LIN {X 0,Y 488.687,Z 319.919,A -85,B 0,C 180,E1 -6521.601,E2 -6521.601} C_VEL
LIN {X 0,Y 488.693,Z 319.925,A -85,B 0,C 180,E1 -6524.803,E2 -6524.803} C_VEL
LIN {X 0,Y 488.728,Z 319.952,A -85,B 0,C 180,E1 -6527.596,E2 -6527.596} C_VEL
LIN {X 0,Y 492.392,Z 332.248,A -85,B 0,C 180,E1 -6530.421,E2 -6530.421} C_VEL
LIN {X 0,Y 495.369,Z 342.536,A -85,B 0,C 180,E1 -6532.607,E2 -6532.607} C_VEL
LIN {X 0,Y 496.704,Z 348.362,A -85,B 0,C 180,E1 -6533.756,E2 -6533.756} C_VEL
LIN {X 0,Y 495.507,Z 364.581,A -85,B 0,C 180,E1 -6536.42,E2 -6536.42} C_VEL
LIN {X 0,Y 494.27,Z 383.903,A -85,B 0,C 180,E1 -6539.451,E2 -6539.451} C_VEL
LIN {X 0,Y 493.327,Z 401.965,A -85,B 0,C 180,E1 -6542.171,E2 -6542.171} C_VEL
LIN {X 0,Y 492.268,Z 420.732,A -85,B 0,C 180,E1 -6544.998,E2 -6544.998} C_VEL
LIN {X 0,Y 496.9,Z 441.839,A -85,B 0,C 180,E1 -6545.607,E2 -6545.607} C_VEL
LIN {X 0,Y 496.367,Z 458.327,A -85,B 0,C 180,E1 -6546.014,E2 -6546.014} C_VEL
LIN {X 0,Y 495.765,Z 473.338,A -85,B 0,C 180,E1 -6546.533,E2 -6546.533} C_VEL
LIN {X 0,Y 495.092,Z 488.171,A -85,B 0,C 180,E1 -6547.191,E2 -6547.191} C_VEL
LIN {X 0,Y 494.154,Z 504.481,A -85,B 0,C 180,E1 -6548.107,E2 -6548.107} C_VEL
LIN {X 0,Y 493.218,Z 519.301,A -85,B 0,C 180,E1 -6549.134,E2 -6549.134} C_VEL
LIN {X 0,Y 492.292,Z 533.052,A -85,B 0,C 180,E1 -6550.275,E2 -6550.275} C_VEL
LIN {X 0,Y 491.438,Z 545.141,A -85,B 0,C 180,E1 -6551.449,E2 -6551.449} C_VEL
LIN {X 0,Y 490.654,Z 556.299,A -85,B 0,C 180,E1 -6552.712,E2 -6552.712} C_VEL
LIN {X 0,Y 489.963,Z 567.437,A -85,B 0,C 180,E1 -6554.187,E2 -6554.187} C_VEL
LIN {X 0,Y 489.276,Z 578.223,A -85,B 0,C 180,E1 -6555.868,E2 -6555.868} C_VEL
LIN {X 0,Y 488.782,Z 587.283,A -85,B 0,C 180,E1 -6557.547,E2 -6557.547} C_VEL
LIN {X 0,Y 488.439,Z 594.861,A -85,B 0,C 180,E1 -6559.221,E2 -6559.221} C_VEL
LIN {X 0,Y 488.13,Z 602.47,A -85,B 0,C 180,E1 -6561.307,E2 -6561.307} C_VEL
LIN {X 0,Y 488.025,Z 608.25,A -85,B 0,C 180,E1 -6563.387,E2 -6563.387} C_VEL
LIN {X 0,Y 487.908,Z 611.638,A -85,B 0,C 180,E1 -6565.044,E2 -6565.044} C_VEL
LIN {X 0,Y 487.943,Z 614.092,A -85,B 0,C 180,E1 -6566.699,E2 -6566.699} C_VEL
LIN {X 0,Y 487.883,Z 615.48,A -85,B 0,C 180,E1 -6568.351,E2 -6568.351} C_VEL
LIN {X 0,Y 487.814,Z 616,A -85,B 0,C 180,E1 -6570.002,E2 -6570.002} C_VEL
LIN {X 0,Y 487.883,Z 615.477,A -85,B 0,C 180,E1 -6571.653,E2 -6571.653} C_VEL
LIN {X 0,Y 487.945,Z 614.087,A -85,B 0,C 180,E1 -6573.305,E2 -6573.305} C_VEL
LIN {X 0,Y 487.909,Z 611.631,A -85,B 0,C 180,E1 -6574.96,E2 -6574.96} C_VEL
LIN {X 0,Y 488.029,Z 608.246,A -85,B 0,C 180,E1 -6576.617,E2 -6576.617} C_VEL
LIN {X 0,Y 488.124,Z 602.462,A -85,B 0,C 180,E1 -6578.697,E2 -6578.697} C_VEL
LIN {X 0,Y 488.436,Z 594.848,A -85,B 0,C 180,E1 -6580.783,E2 -6580.783} C_VEL
LIN {X 0,Y 488.826,Z 586.246,A -85,B 0,C 180,E1 -6582.667,E2 -6582.667} C_VEL
LIN {X 0,Y 489.349,Z 576.967,A -85,B 0,C 180,E1 -6584.346,E2 -6584.346} C_VEL
LIN {X 0,Y 489.93,Z 567.409,A -85,B 0,C 180,E1 -6585.818,E2 -6585.818} C_VEL
LIN {X 0,Y 490.661,Z 556.269,A -85,B 0,C 180,E1 -6587.292,E2 -6587.292} C_VEL
LIN {X 0,Y 491.499,Z 544.123,A -85,B 0,C 180,E1 -6588.661,E2 -6588.661} C_VEL
LIN {X 0,Y 492.423,Z 530.761,A -85,B 0,C 180,E1 -6589.932,E2 -6589.932} C_VEL
LIN {X 0,Y 493.327,Z 517.822,A -85,B 0,C 180,E1 -6590.975,E2 -6590.975} C_VEL
LIN {X 0,Y 494.159,Z 504.385,A -85,B 0,C 180,E1 -6591.899,E2 -6591.899} C_VEL
LIN {X 0,Y 495.108,Z 488.383,A -85,B 0,C 180,E1 -6592.796,E2 -6592.796} C_VEL
LIN {X 0,Y 495.69,Z 475.201,A -85,B 0,C 180,E1 -6593.392,E2 -6593.392} C_VEL
LIN {X 0,Y 496.355,Z 458.459,A -85,B 0,C 180,E1 -6593.983,E2 -6593.983} C_VEL
LIN {X 0,Y 496.893,Z 442.168,A -85,B 0,C 180,E1 -6594.387,E2 -6594.387} C_VEL
LIN {X 0,Y 493.328,Z 425.29,A -85,B 0,C 180,E1 -6594.865,E2 -6594.865} C_VEL
LIN {X 0,Y 492.313,Z 420.685,A -85,B 0,C 180,E1 -6595.006,E2 -6595.006} C_VEL
LIN {X 0,Y 493.312,Z 402.026,A -85,B 0,C 180,E1 -6597.821,E2 -6597.821} C_VEL
LIN {X 0,Y 494.313,Z 382.243,A -85,B 0,C 180,E1 -6600.788,E2 -6600.788} C_VEL
LIN {X 0,Y 495.292,Z 365.983,A -85,B 0,C 180,E1 -6603.29,E2 -6603.29} C_VEL
LIN {X 0,Y 496.841,Z 349.707,A -85,B 0,C 180,E1 -6606.095,E2 -6606.095} C_VEL
LIN {X 0,Y 496.561,Z 346.659,A -85,B 0,C 180,E1 -6606.719,E2 -6606.719} C_VEL
LIN {X 0,Y 494.656,Z 338.928,A -85,B 0,C 180,E1 -6608.609,E2 -6608.609} C_VEL
LIN {X 0,Y 492.734,Z 332.835,A -85,B 0,C 180,E1 -6610.481,E2 -6610.481} C_VEL
LIN {X 0,Y 491.301,Z 328.379,A -85,B 0,C 180,E1 -6612.249,E2 -6612.249} C_VEL
LIN {X 0,Y 490.173,Z 324.874,A -85,B 0,C 180,E1 -6614.202,E2 -6614.202} C_VEL
LIN {X 0,Y 489.577,Z 323.156,A -85,B 0,C 180,E1 -6615.872,E2 -6615.872} C_VEL
LIN {X 0,Y 489.411,Z 322.532,A -85,B 0,C 180,E1 -6617.552,E2 -6617.552} C_VEL
LIN {X 0,Y 489.532,Z 323.246,A -85,B 0,C 180,E1 -6619.545,E2 -6619.545} C_VEL
LIN {X 0,Y 489.855,Z 324.388,A -85,B 0,C 180,E1 -6620.856,E2 -6620.856} C_VEL
LIN {X 0,Y 490.458,Z 327.705,A -85,B 0,C 180,E1 -6623.366,E2 -6623.366} C_VEL
LIN {X 0,Y 490.697,Z 330.547,A -85,B 0,C 180,E1 -6625.048,E2 -6625.048} C_VEL
LIN {X 0,Y 490.306,Z 335.636,A -85,B 0,C 180,E1 -6627.749,E2 -6627.749} C_VEL
LIN {X 0,Y 489.938,Z 341.889,A -85,B 0,C 180,E1 -6631.05,E2 -6631.05} C_VEL
LIN {X 0,Y 489.753,Z 346.67,A -85,B 0,C 180,E1 -6633.586,E2 -6633.586} C_VEL
LIN {X 0,Y 489.517,Z 352.555,A -85,B 0,C 180,E1 -6636.76,E2 -6636.76} C_VEL
LIN {X 0,Y 489.316,Z 358.293,A -85,B 0,C 180,E1 -6639.836,E2 -6639.836} C_VEL
LIN {X 0,Y 489.109,Z 363.152,A -85,B 0,C 180,E1 -6642.438,E2 -6642.438} C_VEL
LIN {X 0,Y 489.022,Z 367.71,A -85,B 0,C 180,E1 -6644.846,E2 -6644.846} C_VEL
LIN {X 0,Y 492.349,Z 378.298,A -85,B 0,C 180,E1 -6645.323,E2 -6645.323} C_VEL
LIN {X 0,Y 491.939,Z 392.152,A -85,B 0,C 180,E1 -6645.892,E2 -6645.892} C_VEL
LIN {X 0,Y 491.362,Z 405.497,A -85,B 0,C 180,E1 -6646.634,E2 -6646.634} C_VEL
LIN {X 0,Y 490.964,Z 417.712,A -85,B 0,C 180,E1 -6647.515,E2 -6647.515} C_VEL
LIN {X 0,Y 490.431,Z 428.93,A -85,B 0,C 180,E1 -6648.532,E2 -6648.532} C_VEL
LIN {X 0,Y 490.077,Z 439.066,A -85,B 0,C 180,E1 -6649.674,E2 -6649.674} C_VEL
LIN {X 0,Y 489.619,Z 447.947,A -85,B 0,C 180,E1 -6650.916,E2 -6650.916} C_VEL
LIN {X 0,Y 489.345,Z 454.492,A -85,B 0,C 180,E1 -6652.044,E2 -6652.044} C_VEL
LIN {X 0,Y 489.014,Z 460.816,A -85,B 0,C 180,E1 -6653.398,E2 -6653.398} C_VEL
LIN {X 0,Y 488.814,Z 465.319,A -85,B 0,C 180,E1 -6654.638,E2 -6654.638} C_VEL
LIN {X 0,Y 488.754,Z 468.722,A -85,B 0,C 180,E1 -6655.877,E2 -6655.877} C_VEL
LIN {X 0,Y 488.686,Z 470.465,A -85,B 0,C 180,E1 -6656.703,E2 -6656.703} C_VEL
LIN {X 0,Y 488.565,Z 471.782,A -85,B 0,C 180,E1 -6657.527,E2 -6657.527} C_VEL
LIN {X 0,Y 488.377,Z 473.181,A -85,B 0,C 180,E1 -6659.176,E2 -6659.176} C_VEL
LIN {X 0,Y 488.357,Z 473.297,A -85,B 0,C 180,E1 -6660,E2 -6660} C_VEL
LIN {X 0,Y 488.366,Z 473.016,A -85,B 0,C 180,E1 -6660.825,E2 -6660.825} C_VEL
LIN {X 0,Y 488.43,Z 472.307,A -85,B 0,C 180,E1 -6661.649,E2 -6661.649} C_VEL
LIN {X 0,Y 488.431,Z 471.22,A -85,B 0,C 180,E1 -6662.474,E2 -6662.474} C_VEL
LIN {X 0,Y 488.547,Z 469.723,A -85,B 0,C 180,E1 -6663.299,E2 -6663.299} C_VEL
LIN {X 0,Y 488.513,Z 466.692,A -85,B 0,C 180,E1 -6664.539,E2 -6664.539} C_VEL
LIN {X 0,Y 488.635,Z 462.622,A -85,B 0,C 180,E1 -6665.779,E2 -6665.779} C_VEL
LIN {X 0,Y 488.827,Z 456.426,A -85,B 0,C 180,E1 -6667.232,E2 -6667.232} C_VEL
LIN {X 0,Y 489.088,Z 449.68,A -85,B 0,C 180,E1 -6668.47,E2 -6668.47} C_VEL
LIN {X 0,Y 489.342,Z 441.317,A -85,B 0,C 180,E1 -6669.716,E2 -6669.716} C_VEL
LIN {X 0,Y 489.638,Z 432.812,A -85,B 0,C 180,E1 -6670.754,E2 -6670.754} C_VEL
LIN {X 0,Y 490.038,Z 422.438,A -85,B 0,C 180,E1 -6671.793,E2 -6671.793} C_VEL
LIN {X 0,Y 490.401,Z 411.409,A -85,B 0,C 180,E1 -6672.684,E2 -6672.684} C_VEL
LIN {X 0,Y 490.868,Z 399.455,A -85,B 0,C 180,E1 -6673.454,E2 -6673.454} C_VEL
LIN {X 0,Y 491.139,Z 386.946,A -85,B 0,C 180,E1 -6674.08,E2 -6674.08} C_VEL
LIN {X 0,Y 491.244,Z 376.285,A -85,B 0,C 180,E1 -6674.486,E2 -6674.486} C_VEL
LIN {X 0,Y 488.33,Z 363.648,A -85,B 0,C 180,E1 -6674.934,E2 -6674.934} C_VEL
LIN {X 0,Y 488.388,Z 356.44,A -85,B 0,C 180,E1 -6678.457,E2 -6678.457} C_VEL
LIN {X 0,Y 488.55,Z 349.357,A -85,B 0,C 180,E1 -6681.964,E2 -6681.964} C_VEL
LIN {X 0,Y 488.661,Z 343.202,A -85,B 0,C 180,E1 -6685.029,E2 -6685.029} C_VEL
LIN {X 0,Y 488.725,Z 338.504,A -85,B 0,C 180,E1 -6687.398,E2 -6687.398} C_VEL
LIN {X 0,Y 488.885,Z 332.597,A -85,B 0,C 180,E1 -6690.396,E2 -6690.396} C_VEL
LIN {X 0,Y 489.043,Z 326.458,A -85,B 0,C 180,E1 -6693.537,E2 -6693.537} C_VEL
LIN {X 0,Y 488.964,Z 321.505,A -85,B 0,C 180,E1 -6696.108,E2 -6696.108} C_VEL
LIN {X 0,Y 488.712,Z 319.925,A -85,B 0,C 180,E1 -6697.052,E2 -6697.052} C_VEL
LIN {X 0,Y 488.727,Z 319.923,A -85,B 0,C 180,E1 -6700.344,E2 -6700.344} C_VEL
LIN {X 0,Y 488.686,Z 319.926,A -85,B 0,C 180,E1 -6703.655,E2 -6703.655} C_VEL
LIN {X 0,Y 488.685,Z 319.927,A -85,B 0,C 180,E1 -6706.344,E2 -6706.344} C_VEL
LIN {X 0,Y 488.712,Z 319.922,A -85,B 0,C 180,E1 -6709.673,E2 -6709.673} C_VEL
LIN {X 0,Y 488.696,Z 319.928,A -85,B 0,C 180,E1 -6712.841,E2 -6712.841} C_VEL
LIN {X 0,Y 488.785,Z 320.145,A -85,B 0,C 180,E1 -6713.49,E2 -6713.49} C_VEL
LIN {X 0,Y 489.294,Z 324.961,A -85,B 0,C 180,E1 -6715.451,E2 -6715.451} C_VEL
LIN {X 0,Y 489.247,Z 329.472,A -85,B 0,C 180,E1 -6717.377,E2 -6717.377} C_VEL
LIN {X 0,Y 488.584,Z 331.063,A -85,B 0,C 180,E1 -6718.038,E2 -6718.038} C_VEL
LIN {X 0,Y 485.698,Z 333.904,A -85,B 0,C 180,E1 -6719.103,E2 -6719.103} C_VEL
LIN {X 0,Y 483.247,Z 336.161,A -85,B 0,C 180,E1 -6719.961,E2 -6719.961} C_VEL
LIN {X 0,Y 482.19,Z 337.745,A -85,B 0,C 180,E1 -6720.63,E2 -6720.63} C_VEL
LIN {X 0,Y 482.103,Z 338.23,A -85,B 0,C 180,E1 -6720.858,E2 -6720.858} C_VEL
LIN {X 0,Y 481.968,Z 344.726,A -85,B 0,C 180,E1 -6724.057,E2 -6724.057} C_VEL
LIN {X 0,Y 481.938,Z 350.288,A -85,B 0,C 180,E1 -6726.811,E2 -6726.811} C_VEL
LIN {X 0,Y 481.835,Z 355.858,A -85,B 0,C 180,E1 -6729.507,E2 -6729.507} C_VEL
LIN {X 0,Y 481.786,Z 362.714,A -85,B 0,C 180,E1 -6732.598,E2 -6732.598} C_VEL
LIN {X 0,Y 481.935,Z 369.073,A -85,B 0,C 180,E1 -6735.145,E2 -6735.145} C_VEL
LIN {X 0,Y 484.514,Z 378.706,A -85,B 0,C 180,E1 -6735.462,E2 -6735.462} C_VEL
LIN {X 0,Y 484.31,Z 391.761,A -85,B 0,C 180,E1 -6735.931,E2 -6735.931} C_VEL
LIN {X 0,Y 483.99,Z 404.316,A -85,B 0,C 180,E1 -6736.564,E2 -6736.564} C_VEL
LIN {X 0,Y 483.777,Z 415.235,A -85,B 0,C 180,E1 -6737.293,E2 -6737.293} C_VEL
LIN {X 0,Y 483.401,Z 425.434,A -85,B 0,C 180,E1 -6738.148,E2 -6738.148} C_VEL
LIN {X 0,Y 482.991,Z 434.651,A -85,B 0,C 180,E1 -6739.094,E2 -6739.094} C_VEL
LIN {X 0,Y 482.672,Z 443.053,A -85,B 0,C 180,E1 -6740.147,E2 -6740.147} C_VEL
LIN {X 0,Y 482.284,Z 451.234,A -85,B 0,C 180,E1 -6741.408,E2 -6741.408} C_VEL
LIN {X 0,Y 481.965,Z 457.873,A -85,B 0,C 180,E1 -6742.692,E2 -6742.692} C_VEL
LIN {X 0,Y 481.743,Z 463.73,A -85,B 0,C 180,E1 -6744.137,E2 -6744.137} C_VEL
LIN {X 0,Y 481.532,Z 467.616,A -85,B 0,C 180,E1 -6745.394,E2 -6745.394} C_VEL
LIN {X 0,Y 481.453,Z 470.471,A -85,B 0,C 180,E1 -6746.651,E2 -6746.651} C_VEL
LIN {X 0,Y 481.419,Z 471.858,A -85,B 0,C 180,E1 -6747.488,E2 -6747.488} C_VEL
LIN {X 0,Y 481.352,Z 473.433,A -85,B 0,C 180,E1 -6749.161,E2 -6749.161} C_VEL
LIN {X 0,Y 481.337,Z 473.667,A -85,B 0,C 180,E1 -6749.998,E2 -6749.998} C_VEL
LIN {X 0,Y 481.351,Z 473.484,A -85,B 0,C 180,E1 -6750.835,E2 -6750.835} C_VEL
LIN {X 0,Y 481.294,Z 472.929,A -85,B 0,C 180,E1 -6751.671,E2 -6751.671} C_VEL
LIN {X 0,Y 481.558,Z 470.64,A -85,B 0,C 180,E1 -6753.345,E2 -6753.345} C_VEL
LIN {X 0,Y 481.622,Z 467.856,A -85,B 0,C 180,E1 -6754.601,E2 -6754.601} C_VEL
LIN {X 0,Y 481.733,Z 464.067,A -85,B 0,C 180,E1 -6755.859,E2 -6755.859} C_VEL
LIN {X 0,Y 481.879,Z 459.586,A -85,B 0,C 180,E1 -6757.019,E2 -6757.019} C_VEL
LIN {X 0,Y 482.197,Z 452.93,A -85,B 0,C 180,E1 -6758.378,E2 -6758.378} C_VEL
LIN {X 0,Y 482.586,Z 445.185,A -85,B 0,C 180,E1 -6759.639,E2 -6759.639} C_VEL
LIN {X 0,Y 482.9,Z 437.274,A -85,B 0,C 180,E1 -6760.691,E2 -6760.691} C_VEL
LIN {X 0,Y 483.287,Z 427.556,A -85,B 0,C 180,E1 -6761.745,E2 -6761.745} C_VEL
LIN {X 0,Y 483.605,Z 417.954,A -85,B 0,C 180,E1 -6762.589,E2 -6762.589} C_VEL
LIN {X 0,Y 483.943,Z 405.879,A -85,B 0,C 180,E1 -6763.434,E2 -6763.434} C_VEL
LIN {X 0,Y 484.272,Z 393.904,A -85,B 0,C 180,E1 -6764.066,E2 -6764.066} C_VEL
LIN {X 0,Y 484.476,Z 380.633,A -85,B 0,C 180,E1 -6764.57,E2 -6764.57} C_VEL
LIN {X 0,Y 484.196,Z 377.035,A -85,B 0,C 180,E1 -6764.684,E2 -6764.684} C_VEL
LIN {X 0,Y 481.89,Z 368.836,A -85,B 0,C 180,E1 -6764.974,E2 -6764.974} C_VEL
LIN {X 0,Y 481.776,Z 361.933,A -85,B 0,C 180,E1 -6767.836,E2 -6767.836} C_VEL
LIN {X 0,Y 481.85,Z 354.941,A -85,B 0,C 180,E1 -6771.017,E2 -6771.017} C_VEL
LIN {X 0,Y 481.946,Z 348.668,A -85,B 0,C 180,E1 -6774.096,E2 -6774.096} C_VEL
LIN {X 0,Y 482.04,Z 342.372,A -85,B 0,C 180,E1 -6777.206,E2 -6777.206} C_VEL
LIN {X 0,Y 482.189,Z 336.25,A -85,B 0,C 180,E1 -6780.185,E2 -6780.185} C_VEL
LIN {X 0,Y 482.285,Z 329.836,A -85,B 0,C 180,E1 -6783.121,E2 -6783.121} C_VEL
LIN {X 0,Y 482.199,Z 323.807,A -85,B 0,C 180,E1 -6785.658,E2 -6785.658} C_VEL
LIN {X 0,Y 481.7,Z 320.8,A -85,B 0,C 180,E1 -6786.867,E2 -6786.867} C_VEL
LIN {X 0,Y 481.646,Z 320.805,A -85,B 0,C 180,E1 -6789.94,E2 -6789.94} C_VEL
LIN {X 0,Y 481.613,Z 320.808,A -85,B 0,C 180,E1 -6793.144,E2 -6793.144} C_VEL
LIN {X 0,Y 481.644,Z 320.801,A -85,B 0,C 180,E1 -6795.638,E2 -6795.638} C_VEL
LIN {X 0,Y 481.66,Z 320.798,A -85,B 0,C 180,E1 -6798.082,E2 -6798.082} C_VEL
LIN {X 0,Y 481.689,Z 320.794,A -85,B 0,C 180,E1 -6801.142,E2 -6801.142} C_VEL
LIN {X 0,Y 481.648,Z 320.799,A -85,B 0,C 180,E1 -6804.793,E2 -6804.793} C_VEL
LIN {X 0,Y 481.652,Z 320.802,A -85,B 0,C 180,E1 -6807.324,E2 -6807.324} C_VEL
LIN {X 0,Y 481.658,Z 320.796,A -85,B 0,C 180,E1 -6810.257,E2 -6810.257} C_VEL
LIN {X 0,Y 481.731,Z 320.786,A -85,B 0,C 180,E1 -6813.111,E2 -6813.111} C_VEL
LIN {X 0,Y 481.672,Z 320.8,A -85,B 0,C 180,E1 -6815.886,E2 -6815.886} C_VEL
LIN {X 0,Y 481.688,Z 320.795,A -85,B 0,C 180,E1 -6819.023,E2 -6819.023} C_VEL
LIN {X 0,Y 481.682,Z 320.793,A -85,B 0,C 180,E1 -6822.157,E2 -6822.157} C_VEL
LIN {X 0,Y 481.718,Z 320.793,A -85,B 0,C 180,E1 -6824.775,E2 -6824.775} C_VEL
LIN {X 0,Y 481.777,Z 320.787,A -85,B 0,C 180,E1 -6828.215,E2 -6828.215} C_VEL
LIN {X 0,Y 481.747,Z 320.786,A -85,B 0,C 180,E1 -6831.611,E2 -6831.611} C_VEL
LIN {X 0,Y 481.797,Z 320.779,A -85,B 0,C 180,E1 -6834.139,E2 -6834.139} C_VEL
LIN {X 0,Y 481.898,Z 320.77,A -85,B 0,C 180,E1 -6837.492,E2 -6837.492} C_VEL
LIN {X 0,Y 481.902,Z 320.766,A -85,B 0,C 180,E1 -6840.835,E2 -6840.835} C_VEL
LIN {X 0,Y 481.912,Z 320.771,A -85,B 0,C 180,E1 -6842.507,E2 -6842.507} C_VEL
LIN {X 0,Y 481.809,Z 320.785,A -85,B 0,C 180,E1 -6845.86,E2 -6845.86} C_VEL
LIN {X 0,Y 481.739,Z 320.788,A -85,B 0,C 180,E1 -6848.388,E2 -6848.388} C_VEL
LIN {X 0,Y 481.772,Z 320.785,A -85,B 0,C 180,E1 -6851.784,E2 -6851.784} C_VEL
LIN {X 0,Y 481.718,Z 320.791,A -85,B 0,C 180,E1 -6855.225,E2 -6855.225} C_VEL
LIN {X 0,Y 481.693,Z 320.794,A -85,B 0,C 180,E1 -6858.722,E2 -6858.722} C_VEL
LIN {X 0,Y 481.654,Z 320.803,A -85,B 0,C 180,E1 -6861.394,E2 -6861.394} C_VEL
LIN {X 0,Y 481.665,Z 320.797,A -85,B 0,C 180,E1 -6864.113,E2 -6864.113} C_VEL
LIN {X 0,Y 481.722,Z 320.792,A -85,B 0,C 180,E1 -6867.14,E2 -6867.14} C_VEL
LIN {X 0,Y 481.655,Z 320.799,A -85,B 0,C 180,E1 -6869.742,E2 -6869.742} C_VEL
LIN {X 0,Y 481.651,Z 320.8,A -85,B 0,C 180,E1 -6872.675,E2 -6872.675} C_VEL
LIN {X 0,Y 481.623,Z 320.807,A -85,B 0,C 180,E1 -6875.71,E2 -6875.71} C_VEL
LIN {X 0,Y 481.651,Z 320.802,A -85,B 0,C 180,E1 -6878.861,E2 -6878.861} C_VEL
LIN {X 0,Y 481.632,Z 320.799,A -85,B 0,C 180,E1 -6881.915,E2 -6881.915} C_VEL
LIN {X 0,Y 481.641,Z 320.805,A -85,B 0,C 180,E1 -6884.459,E2 -6884.459} C_VEL
LIN {X 0,Y 481.701,Z 320.949,A -85,B 0,C 180,E1 -6886.997,E2 -6886.997} C_VEL
LIN {X 0,Y 484.936,Z 331.574,A -85,B 0,C 180,E1 -6889.539,E2 -6889.539} C_VEL
LIN {X 0,Y 488.601,Z 344.148,A -85,B 0,C 180,E1 -6892.289,E2 -6892.289} C_VEL
LIN {X 0,Y 490.108,Z 350.895,A -85,B 0,C 180,E1 -6893.648,E2 -6893.648} C_VEL
LIN {X 0,Y 488.612,Z 369.086,A -85,B 0,C 180,E1 -6896.672,E2 -6896.672} C_VEL
LIN {X 0,Y 487.34,Z 388.12,A -85,B 0,C 180,E1 -6899.689,E2 -6899.689} C_VEL
LIN {X 0,Y 486.277,Z 407.911,A -85,B 0,C 180,E1 -6902.689,E2 -6902.689} C_VEL
LIN {X 0,Y 485.554,Z 420.739,A -85,B 0,C 180,E1 -6904.629,E2 -6904.629} C_VEL
LIN {X 0,Y 490.394,Z 442.388,A -85,B 0,C 180,E1 -6905.272,E2 -6905.272} C_VEL
LIN {X 0,Y 489.844,Z 459.443,A -85,B 0,C 180,E1 -6905.709,E2 -6905.709} C_VEL
LIN {X 0,Y 489.146,Z 475.3,A -85,B 0,C 180,E1 -6906.281,E2 -6906.281} C_VEL
LIN {X 0,Y 488.382,Z 489.912,A -85,B 0,C 180,E1 -6906.958,E2 -6906.958} C_VEL
LIN {X 0,Y 487.538,Z 504.667,A -85,B 0,C 180,E1 -6907.806,E2 -6907.806} C_VEL
LIN {X 0,Y 486.544,Z 519.299,A -85,B 0,C 180,E1 -6908.834,E2 -6908.834} C_VEL
LIN {X 0,Y 485.608,Z 532.128,A -85,B 0,C 180,E1 -6909.905,E2 -6909.905} C_VEL
LIN {X 0,Y 484.731,Z 544.166,A -85,B 0,C 180,E1 -6911.073,E2 -6911.073} C_VEL
LIN {X 0,Y 483.78,Z 556.299,A -85,B 0,C 180,E1 -6912.458,E2 -6912.458} C_VEL
LIN {X 0,Y 483.031,Z 567.437,A -85,B 0,C 180,E1 -6913.954,E2 -6913.954} C_VEL
LIN {X 0,Y 482.3,Z 578.222,A -85,B 0,C 180,E1 -6915.66,E2 -6915.66} C_VEL
LIN {X 0,Y 481.741,Z 587.284,A -85,B 0,C 180,E1 -6917.362,E2 -6917.362} C_VEL
LIN {X 0,Y 481.413,Z 594.86,A -85,B 0,C 180,E1 -6919.062,E2 -6919.062} C_VEL
LIN {X 0,Y 481.063,Z 602.47,A -85,B 0,C 180,E1 -6921.178,E2 -6921.178} C_VEL
LIN {X 0,Y 480.948,Z 608.25,A -85,B 0,C 180,E1 -6923.289,E2 -6923.289} C_VEL
LIN {X 0,Y 480.834,Z 611.638,A -85,B 0,C 180,E1 -6924.971,E2 -6924.971} C_VEL
LIN {X 0,Y 480.849,Z 614.092,A -85,B 0,C 180,E1 -6926.651,E2 -6926.651} C_VEL
LIN {X 0,Y 480.784,Z 615.48,A -85,B 0,C 180,E1 -6928.327,E2 -6928.327} C_VEL
LIN {X 0,Y 480.738,Z 616,A -85,B 0,C 180,E1 -6930.002,E2 -6930.002} C_VEL
LIN {X 0,Y 480.784,Z 615.477,A -85,B 0,C 180,E1 -6931.677,E2 -6931.677} C_VEL
LIN {X 0,Y 480.85,Z 614.087,A -85,B 0,C 180,E1 -6933.354,E2 -6933.354} C_VEL
LIN {X 0,Y 480.836,Z 611.631,A -85,B 0,C 180,E1 -6935.033,E2 -6935.033} C_VEL
LIN {X 0,Y 480.952,Z 608.247,A -85,B 0,C 180,E1 -6936.715,E2 -6936.715} C_VEL
LIN {X 0,Y 481.058,Z 602.462,A -85,B 0,C 180,E1 -6938.826,E2 -6938.826} C_VEL
LIN {X 0,Y 481.402,Z 594.848,A -85,B 0,C 180,E1 -6940.942,E2 -6940.942} C_VEL
LIN {X 0,Y 481.824,Z 586.247,A -85,B 0,C 180,E1 -6942.854,E2 -6942.854} C_VEL
LIN {X 0,Y 482.368,Z 576.967,A -85,B 0,C 180,E1 -6944.558,E2 -6944.558} C_VEL
LIN {X 0,Y 483,Z 567.409,A -85,B 0,C 180,E1 -6946.051,E2 -6946.051} C_VEL
LIN {X 0,Y 483.786,Z 556.269,A -85,B 0,C 180,E1 -6947.546,E2 -6947.546} C_VEL
LIN {X 0,Y 484.705,Z 544.122,A -85,B 0,C 180,E1 -6948.933,E2 -6948.933} C_VEL
LIN {X 0,Y 485.671,Z 530.857,A -85,B 0,C 180,E1 -6950.212,E2 -6950.212} C_VEL
LIN {X 0,Y 486.729,Z 516.394,A -85,B 0,C 180,E1 -6951.384,E2 -6951.384} C_VEL
LIN {X 0,Y 487.643,Z 503.092,A -85,B 0,C 180,E1 -6952.289,E2 -6952.289} C_VEL
LIN {X 0,Y 488.535,Z 488.381,A -85,B 0,C 180,E1 -6953.12,E2 -6953.12} C_VEL
LIN {X 0,Y 489.187,Z 475.201,A -85,B 0,C 180,E1 -6953.722,E2 -6953.722} C_VEL
LIN {X 0,Y 489.855,Z 459.341,A -85,B 0,C 180,E1 -6954.294,E2 -6954.294} C_VEL
LIN {X 0,Y 490.371,Z 443.722,A -85,B 0,C 180,E1 -6954.698,E2 -6954.698} C_VEL
LIN {X 0,Y 489.839,Z 439.91,A -85,B 0,C 180,E1 -6954.805,E2 -6954.805} C_VEL
LIN {X 0,Y 485.581,Z 420.702,A -85,B 0,C 180,E1 -6955.375,E2 -6955.375} C_VEL
LIN {X 0,Y 486.361,Z 404.997,A -85,B 0,C 180,E1 -6957.721,E2 -6957.721} C_VEL
LIN {X 0,Y 487.052,Z 391.301,A -85,B 0,C 180,E1 -6959.748,E2 -6959.748} C_VEL
LIN {X 0,Y 488.439,Z 369.736,A -85,B 0,C 180,E1 -6963.147,E2 -6963.147} C_VEL
LIN {X 0,Y 489.905,Z 354.515,A -85,B 0,C 180,E1 -6965.775,E2 -6965.775} C_VEL
LIN {X 0,Y 490.21,Z 350.269,A -85,B 0,C 180,E1 -6966.597,E2 -6966.597} C_VEL
LIN {X 0,Y 488.486,Z 342.788,A -85,B 0,C 180,E1 -6968.431,E2 -6968.431} C_VEL
LIN {X 0,Y 486.344,Z 335.866,A -85,B 0,C 180,E1 -6970.564,E2 -6970.564} C_VEL
LIN {X 0,Y 484.928,Z 331.462,A -85,B 0,C 180,E1 -6972.343,E2 -6972.343} C_VEL
LIN {X 0,Y 483.912,Z 328.176,A -85,B 0,C 180,E1 -6974.198,E2 -6974.198} C_VEL
LIN {X 0,Y 483.298,Z 326.493,A -85,B 0,C 180,E1 -6975.733,E2 -6975.733} C_VEL
LIN {X 0,Y 483.114,Z 325.812,A -85,B 0,C 180,E1 -6976.865,E2 -6976.865} C_VEL
LIN {X 0,Y 483.014,Z 325.651,A -85,B 0,C 180,E1 -6977.986,E2 -6977.986} C_VEL
LIN {X 0,Y 483.172,Z 326.576,A -85,B 0,C 180,E1 -6980.208,E2 -6980.208} C_VEL
LIN {X 0,Y 483.566,Z 328.817,A -85,B 0,C 180,E1 -6982.381,E2 -6982.381} C_VEL
LIN {X 0,Y 483.943,Z 331.868,A -85,B 0,C 180,E1 -6984.487,E2 -6984.487} C_VEL
LIN {X 0,Y 483.737,Z 335.341,A -85,B 0,C 180,E1 -6986.49,E2 -6986.49} C_VEL
LIN {X 0,Y 483.147,Z 342.416,A -85,B 0,C 180,E1 -6990.359,E2 -6990.359} C_VEL
LIN {X 0,Y 482.872,Z 347.642,A -85,B 0,C 180,E1 -6993.18,E2 -6993.18} C_VEL
LIN {X 0,Y 482.651,Z 352.751,A -85,B 0,C 180,E1 -6995.939,E2 -6995.939} C_VEL
LIN {X 0,Y 482.478,Z 357.918,A -85,B 0,C 180,E1 -6998.791,E2 -6998.791} C_VEL
LIN {X 0,Y 482.256,Z 362.567,A -85,B 0,C 180,E1 -7001.311,E2 -7001.311} C_VEL
LIN {X 0,Y 482.107,Z 368.73,A -85,B 0,C 180,E1 -7004.538,E2 -7004.538} C_VEL
LIN {X 0,Y 485.615,Z 379.619,A -85,B 0,C 180,E1 -7005.061,E2 -7005.061} C_VEL
LIN {X 0,Y 485.266,Z 393.198,A -85,B 0,C 180,E1 -7005.64,E2 -7005.64} C_VEL
LIN {X 0,Y 484.691,Z 405.834,A -85,B 0,C 180,E1 -7006.351,E2 -7006.351} C_VEL
LIN {X 0,Y 484.232,Z 418.091,A -85,B 0,C 180,E1 -7007.239,E2 -7007.239} C_VEL
LIN {X 0,Y 483.759,Z 428.36,A -85,B 0,C 180,E1 -7008.159,E2 -7008.159} C_VEL
LIN {X 0,Y 483.314,Z 438.752,A -85,B 0,C 180,E1 -7009.316,E2 -7009.316} C_VEL
LIN {X 0,Y 482.831,Z 447.947,A -85,B 0,C 180,E1 -7010.576,E2 -7010.576} C_VEL
LIN {X 0,Y 482.466,Z 455.669,A -85,B 0,C 180,E1 -7011.905,E2 -7011.905} C_VEL
LIN {X 0,Y 482.081,Z 462.108,A -85,B 0,C 180,E1 -7013.303,E2 -7013.303} C_VEL
LIN {X 0,Y 481.874,Z 466.596,A -85,B 0,C 180,E1 -7014.56,E2 -7014.56} C_VEL
LIN {X 0,Y 481.796,Z 469.986,A -85,B 0,C 180,E1 -7015.818,E2 -7015.818} C_VEL
LIN {X 0,Y 481.718,Z 471.714,A -85,B 0,C 180,E1 -7016.655,E2 -7016.655} C_VEL
LIN {X 0,Y 481.581,Z 473.018,A -85,B 0,C 180,E1 -7017.491,E2 -7017.491} C_VEL
LIN {X 0,Y 481.382,Z 474.388,A -85,B 0,C 180,E1 -7019.164,E2 -7019.164} C_VEL
LIN {X 0,Y 481.358,Z 474.487,A -85,B 0,C 180,E1 -7020,E2 -7020} C_VEL
LIN {X 0,Y 481.364,Z 474.18,A -85,B 0,C 180,E1 -7020.837,E2 -7020.837} C_VEL
LIN {X 0,Y 481.431,Z 473.445,A -85,B 0,C 180,E1 -7021.673,E2 -7021.673} C_VEL
LIN {X 0,Y 481.429,Z 472.338,A -85,B 0,C 180,E1 -7022.51,E2 -7022.51} C_VEL
LIN {X 0,Y 481.555,Z 470.819,A -85,B 0,C 180,E1 -7023.347,E2 -7023.347} C_VEL
LIN {X 0,Y 481.512,Z 467.75,A -85,B 0,C 180,E1 -7024.605,E2 -7024.605} C_VEL
LIN {X 0,Y 481.667,Z 463.634,A -85,B 0,C 180,E1 -7025.863,E2 -7025.863} C_VEL
LIN {X 0,Y 481.858,Z 457.367,A -85,B 0,C 180,E1 -7027.34,E2 -7027.34} C_VEL
LIN {X 0,Y 482.137,Z 450.586,A -85,B 0,C 180,E1 -7028.593,E2 -7028.593} C_VEL
LIN {X 0,Y 482.405,Z 442.185,A -85,B 0,C 180,E1 -7029.857,E2 -7029.857} C_VEL
LIN {X 0,Y 482.733,Z 433.643,A -85,B 0,C 180,E1 -7030.91,E2 -7030.91} C_VEL
LIN {X 0,Y 483.143,Z 423.235,A -85,B 0,C 180,E1 -7031.964,E2 -7031.964} C_VEL
LIN {X 0,Y 483.587,Z 411.132,A -85,B 0,C 180,E1 -7032.945,E2 -7032.945} C_VEL
LIN {X 0,Y 484.032,Z 400.257,A -85,B 0,C 180,E1 -7033.648,E2 -7033.648} C_VEL
LIN {X 0,Y 484.323,Z 387.847,A -85,B 0,C 180,E1 -7034.282,E2 -7034.282} C_VEL
LIN {X 0,Y 484.422,Z 377.335,A -85,B 0,C 180,E1 -7034.695,E2 -7034.695} C_VEL
LIN {X 0,Y 481.296,Z 364.011,A -85,B 0,C 180,E1 -7035.185,E2 -7035.185} C_VEL
LIN {X 0,Y 481.361,Z 356.8,A -85,B 0,C 180,E1 -7038.736,E2 -7038.736} C_VEL
LIN {X 0,Y 481.455,Z 351.417,A -85,B 0,C 180,E1 -7041.404,E2 -7041.404} C_VEL
LIN {X 0,Y 481.557,Z 346.005,A -85,B 0,C 180,E1 -7044.12,E2 -7044.12} C_VEL
LIN {X 0,Y 481.716,Z 340.045,A -85,B 0,C 180,E1 -7047.13,E2 -7047.13} C_VEL
LIN {X 0,Y 481.83,Z 334.943,A -85,B 0,C 180,E1 -7049.731,E2 -7049.731} C_VEL
LIN {X 0,Y 481.948,Z 329.267,A -85,B 0,C 180,E1 -7052.654,E2 -7052.654} C_VEL
LIN {X 0,Y 482.032,Z 324.239,A -85,B 0,C 180,E1 -7055.265,E2 -7055.265} C_VEL
LIN {X 0,Y 481.674,Z 320.802,A -85,B 0,C 180,E1 -7057.135,E2 -7057.135} C_VEL
LIN {X 0,Y 481.666,Z 320.804,A -85,B 0,C 180,E1 -7059.942,E2 -7059.942} C_VEL
LIN {X 0,Y 481.636,Z 320.804,A -85,B 0,C 180,E1 -7063.146,E2 -7063.146} C_VEL
LIN {X 0,Y 481.661,Z 320.802,A -85,B 0,C 180,E1 -7065.641,E2 -7065.641} C_VEL
LIN {X 0,Y 481.657,Z 320.804,A -85,B 0,C 180,E1 -7068.957,E2 -7068.957} C_VEL
LIN {X 0,Y 481.662,Z 320.804,A -85,B 0,C 180,E1 -7071.992,E2 -7071.992} C_VEL
LIN {X 0,Y 481.689,Z 320.885,A -85,B 0,C 180,E1 -7073.257,E2 -7073.257} C_VEL
LIN {X 0,Y 482.223,Z 324.412,A -85,B 0,C 180,E1 -7074.702,E2 -7074.702} C_VEL
LIN {X 0,Y 482.255,Z 329.554,A -85,B 0,C 180,E1 -7076.872,E2 -7076.872} C_VEL
LIN {X 0,Y 482.149,Z 336.026,A -85,B 0,C 180,E1 -7079.807,E2 -7079.807} C_VEL
LIN {X 0,Y 482.103,Z 338.23,A -85,B 0,C 180,E1 -7080.858,E2 -7080.858} C_VEL
LIN {X 0,Y 481.423,Z 339.742,A -85,B 0,C 180,E1 -7081.531,E2 -7081.531} C_VEL
LIN {X 0,Y 478.526,Z 342.463,A -85,B 0,C 180,E1 -7082.615,E2 -7082.615} C_VEL
LIN {X 0,Y 476.086,Z 344.651,A -85,B 0,C 180,E1 -7083.488,E2 -7083.488} C_VEL
LIN {X 0,Y 475.051,Z 346.203,A -85,B 0,C 180,E1 -7084.167,E2 -7084.167} C_VEL
LIN {X 0,Y 474.974,Z 346.687,A -85,B 0,C 180,E1 -7084.399,E2 -7084.399} C_VEL
LIN {X 0,Y 474.913,Z 352.701,A -85,B 0,C 180,E1 -7087.369,E2 -7087.369} C_VEL
LIN {X 0,Y 474.834,Z 358.476,A -85,B 0,C 180,E1 -7090.096,E2 -7090.096} C_VEL
LIN {X 0,Y 474.847,Z 364.57,A -85,B 0,C 180,E1 -7092.78,E2 -7092.78} C_VEL
LIN {X 0,Y 474.936,Z 369.794,A -85,B 0,C 180,E1 -7094.907,E2 -7094.907} C_VEL
LIN {X 0,Y 477.709,Z 379.759,A -85,B 0,C 180,E1 -7095.251,E2 -7095.251} C_VEL
LIN {X 0,Y 477.496,Z 392.817,A -85,B 0,C 180,E1 -7095.726,E2 -7095.726} C_VEL
LIN {X 0,Y 477.157,Z 405.38,A -85,B 0,C 180,E1 -7096.368,E2 -7096.368} C_VEL
LIN {X 0,Y 476.941,Z 416.294,A -85,B 0,C 180,E1 -7097.108,E2 -7097.108} C_VEL
LIN {X 0,Y 476.541,Z 426.504,A -85,B 0,C 180,E1 -7097.975,E2 -7097.975} C_VEL
LIN {X 0,Y 476.107,Z 435.724,A -85,B 0,C 180,E1 -7098.935,E2 -7098.935} C_VEL
LIN {X 0,Y 475.759,Z 444.128,A -85,B 0,C 180,E1 -7100.003,E2 -7100.003} C_VEL
LIN {X 0,Y 475.351,Z 452.309,A -85,B 0,C 180,E1 -7101.282,E2 -7101.282} C_VEL
LIN {X 0,Y 475.011,Z 458.901,A -85,B 0,C 180,E1 -7102.574,E2 -7102.574} C_VEL
LIN {X 0,Y 474.771,Z 464.805,A -85,B 0,C 180,E1 -7104.05,E2 -7104.05} C_VEL
LIN {X 0,Y 474.535,Z 468.694,A -85,B 0,C 180,E1 -7105.326,E2 -7105.326} C_VEL
LIN {X 0,Y 474.473,Z 471.544,A -85,B 0,C 180,E1 -7106.601,E2 -7106.601} C_VEL
LIN {X 0,Y 474.414,Z 472.934,A -85,B 0,C 180,E1 -7107.451,E2 -7107.451} C_VEL
LIN {X 0,Y 474.344,Z 474.509,A -85,B 0,C 180,E1 -7109.149,E2 -7109.149} C_VEL
LIN {X 0,Y 474.328,Z 474.743,A -85,B 0,C 180,E1 -7109.998,E2 -7109.998} C_VEL
LIN {X 0,Y 474.343,Z 474.56,A -85,B 0,C 180,E1 -7110.847,E2 -7110.847} C_VEL
LIN {X 0,Y 474.427,Z 473.049,A -85,B 0,C 180,E1 -7112.545,E2 -7112.545} C_VEL
LIN {X 0,Y 474.563,Z 471.713,A -85,B 0,C 180,E1 -7113.394,E2 -7113.394} C_VEL
LIN {X 0,Y 474.63,Z 468.929,A -85,B 0,C 180,E1 -7114.669,E2 -7114.669} C_VEL
LIN {X 0,Y 474.76,Z 465.139,A -85,B 0,C 180,E1 -7115.946,E2 -7115.946} C_VEL
LIN {X 0,Y 474.931,Z 460.553,A -85,B 0,C 180,E1 -7117.147,E2 -7117.147} C_VEL
LIN {X 0,Y 475.265,Z 453.999,A -85,B 0,C 180,E1 -7118.502,E2 -7118.502} C_VEL
LIN {X 0,Y 475.669,Z 446.253,A -85,B 0,C 180,E1 -7119.78,E2 -7119.78} C_VEL
LIN {X 0,Y 476.005,Z 438.339,A -85,B 0,C 180,E1 -7120.848,E2 -7120.848} C_VEL
LIN {X 0,Y 476.416,Z 428.618,A -85,B 0,C 180,E1 -7121.916,E2 -7121.916} C_VEL
LIN {X 0,Y 476.762,Z 419.01,A -85,B 0,C 180,E1 -7122.772,E2 -7122.772} C_VEL
LIN {X 0,Y 477.112,Z 406.929,A -85,B 0,C 180,E1 -7123.63,E2 -7123.63} C_VEL
LIN {X 0,Y 477.472,Z 394.936,A -85,B 0,C 180,E1 -7124.271,E2 -7124.271} C_VEL
LIN {X 0,Y 477.681,Z 381.641,A -85,B 0,C 180,E1 -7124.781,E2 -7124.781} C_VEL
LIN {X 0,Y 477.401,Z 378.464,A -85,B 0,C 180,E1 -7124.886,E2 -7124.886} C_VEL
LIN {X 0,Y 474.923,Z 369.781,A -85,B 0,C 180,E1 -7125.199,E2 -7125.199} C_VEL
LIN {X 0,Y 474.814,Z 362.732,A -85,B 0,C 180,E1 -7128.107,E2 -7128.107} C_VEL
LIN {X 0,Y 474.883,Z 355.903,A -85,B 0,C 180,E1 -7131.193,E2 -7131.193} C_VEL
LIN {X 0,Y 474.923,Z 351.022,A -85,B 0,C 180,E1 -7133.547,E2 -7133.547} C_VEL
LIN {X 0,Y 475.001,Z 345.411,A -85,B 0,C 180,E1 -7136.348,E2 -7136.348} C_VEL
LIN {X 0,Y 475.136,Z 339.498,A -85,B 0,C 180,E1 -7139.225,E2 -7139.225} C_VEL
LIN {X 0,Y 475.251,Z 333.241,A -85,B 0,C 180,E1 -7142.162,E2 -7142.162} C_VEL
LIN {X 0,Y 475.331,Z 327.426,A -85,B 0,C 180,E1 -7144.694,E2 -7144.694} C_VEL
LIN {X 0,Y 474.988,Z 323.574,A -85,B 0,C 180,E1 -7146.285,E2 -7146.285} C_VEL
LIN {X 0,Y 474.634,Z 321.679,A -85,B 0,C 180,E1 -7147.107,E2 -7147.107} C_VEL
LIN {X 0,Y 474.601,Z 321.679,A -85,B 0,C 180,E1 -7150.656,E2 -7150.656} C_VEL
LIN {X 0,Y 474.578,Z 321.685,A -85,B 0,C 180,E1 -7153.478,E2 -7153.478} C_VEL
LIN {X 0,Y 474.62,Z 321.677,A -85,B 0,C 180,E1 -7156.512,E2 -7156.512} C_VEL
LIN {X 0,Y 474.625,Z 321.674,A -85,B 0,C 180,E1 -7159.343,E2 -7159.343} C_VEL
LIN {X 0,Y 474.604,Z 321.678,A -85,B 0,C 180,E1 -7161.7,E2 -7161.7} C_VEL
LIN {X 0,Y 474.61,Z 321.676,A -85,B 0,C 180,E1 -7164.724,E2 -7164.724} C_VEL
LIN {X 0,Y 474.615,Z 321.678,A -85,B 0,C 180,E1 -7167.786,E2 -7167.786} C_VEL
LIN {X 0,Y 474.603,Z 321.68,A -85,B 0,C 180,E1 -7170.883,E2 -7170.883} C_VEL
LIN {X 0,Y 474.646,Z 321.667,A -85,B 0,C 180,E1 -7173.627,E2 -7173.627} C_VEL
LIN {X 0,Y 474.632,Z 321.671,A -85,B 0,C 180,E1 -7176.635,E2 -7176.635} C_VEL
LIN {X 0,Y 474.654,Z 321.672,A -85,B 0,C 180,E1 -7179.184,E2 -7179.184} C_VEL
LIN {X 0,Y 474.633,Z 321.673,A -85,B 0,C 180,E1 -7181.883,E2 -7181.883} C_VEL
LIN {X 0,Y 474.675,Z 321.67,A -85,B 0,C 180,E1 -7184.543,E2 -7184.543} C_VEL
LIN {X 0,Y 474.719,Z 321.665,A -85,B 0,C 180,E1 -7188.038,E2 -7188.038} C_VEL
LIN {X 0,Y 474.712,Z 321.661,A -85,B 0,C 180,E1 -7191.486,E2 -7191.486} C_VEL
LIN {X 0,Y 474.759,Z 321.657,A -85,B 0,C 180,E1 -7194.052,E2 -7194.052} C_VEL
LIN {X 0,Y 474.865,Z 321.647,A -85,B 0,C 180,E1 -7197.455,E2 -7197.455} C_VEL
LIN {X 0,Y 474.853,Z 321.644,A -85,B 0,C 180,E1 -7200.848,E2 -7200.848} C_VEL
LIN {X 0,Y 474.879,Z 321.647,A -85,B 0,C 180,E1 -7202.544,E2 -7202.544} C_VEL
LIN {X 0,Y 474.769,Z 321.661,A -85,B 0,C 180,E1 -7205.947,E2 -7205.947} C_VEL
LIN {X 0,Y 474.705,Z 321.664,A -85,B 0,C 180,E1 -7208.514,E2 -7208.514} C_VEL
LIN {X 0,Y 474.715,Z 321.664,A -85,B 0,C 180,E1 -7211.962,E2 -7211.962} C_VEL
LIN {X 0,Y 474.677,Z 321.669,A -85,B 0,C 180,E1 -7215.778,E2 -7215.778} C_VEL
LIN {X 0,Y 474.644,Z 321.672,A -85,B 0,C 180,E1 -7219.011,E2 -7219.011} C_VEL
LIN {X 0,Y 474.621,Z 321.678,A -85,B 0,C 180,E1 -7221.727,E2 -7221.727} C_VEL
LIN {X 0,Y 474.642,Z 321.673,A -85,B 0,C 180,E1 -7224.493,E2 -7224.493} C_VEL
LIN {X 0,Y 474.656,Z 321.671,A -85,B 0,C 180,E1 -7227.335,E2 -7227.335} C_VEL
LIN {X 0,Y 474.582,Z 321.682,A -85,B 0,C 180,E1 -7230.812,E2 -7230.812} C_VEL
LIN {X 0,Y 474.617,Z 321.679,A -85,B 0,C 180,E1 -7233.986,E2 -7233.986} C_VEL
LIN {X 0,Y 474.556,Z 321.685,A -85,B 0,C 180,E1 -7236.902,E2 -7236.902} C_VEL
LIN {X 0,Y 474.607,Z 321.677,A -85,B 0,C 180,E1 -7239.649,E2 -7239.649} C_VEL
LIN {X 0,Y 474.595,Z 321.678,A -85,B 0,C 180,E1 -7242.936,E2 -7242.936} C_VEL
LIN {X 0,Y 474.614,Z 321.681,A -85,B 0,C 180,E1 -7246.17,E2 -7246.17} C_VEL
LIN {X 0,Y 474.611,Z 321.793,A -85,B 0,C 180,E1 -7246.344,E2 -7246.344} C_VEL
LIN {X 0,Y 477.807,Z 332.258,A -85,B 0,C 180,E1 -7248.923,E2 -7248.923} C_VEL
LIN {X 0,Y 481.396,Z 344.48,A -85,B 0,C 180,E1 -7251.693,E2 -7251.693} C_VEL
LIN {X 0,Y 483.464,Z 352.783,A -85,B 0,C 180,E1 -7253.419,E2 -7253.419} C_VEL
LIN {X 0,Y 482.227,Z 367.408,A -85,B 0,C 180,E1 -7255.919,E2 -7255.919} C_VEL
LIN {X 0,Y 480.691,Z 387.726,A -85,B 0,C 180,E1 -7259.225,E2 -7259.225} C_VEL
LIN {X 0,Y 479.607,Z 405.987,A -85,B 0,C 180,E1 -7262.039,E2 -7262.039} C_VEL
LIN {X 0,Y 478.843,Z 420.702,A -85,B 0,C 180,E1 -7264.266,E2 -7264.266} C_VEL
LIN {X 0,Y 483.87,Z 443.265,A -85,B 0,C 180,E1 -7264.936,E2 -7264.936} C_VEL
LIN {X 0,Y 483.341,Z 460.297,A -85,B 0,C 180,E1 -7265.387,E2 -7265.387} C_VEL
LIN {X 0,Y 482.567,Z 476.599,A -85,B 0,C 180,E1 -7265.994,E2 -7265.994} C_VEL
LIN {X 0,Y 481.759,Z 491.141,A -85,B 0,C 180,E1 -7266.693,E2 -7266.693} C_VEL
LIN {X 0,Y 480.828,Z 506.108,A -85,B 0,C 180,E1 -7267.58,E2 -7267.58} C_VEL
LIN {X 0,Y 479.765,Z 520.718,A -85,B 0,C 180,E1 -7268.633,E2 -7268.633} C_VEL
LIN {X 0,Y 478.707,Z 534.411,A -85,B 0,C 180,E1 -7269.821,E2 -7269.821} C_VEL
LIN {X 0,Y 477.661,Z 547.086,A -85,B 0,C 180,E1 -7271.116,E2 -7271.116} C_VEL
LIN {X 0,Y 476.68,Z 559.655,A -85,B 0,C 180,E1 -7272.631,E2 -7272.631} C_VEL
LIN {X 0,Y 475.958,Z 570.361,A -85,B 0,C 180,E1 -7274.149,E2 -7274.149} C_VEL
LIN {X 0,Y 475.155,Z 580.676,A -85,B 0,C 180,E1 -7275.877,E2 -7275.877} C_VEL
LIN {X 0,Y 474.674,Z 589.055,A -85,B 0,C 180,E1 -7277.554,E2 -7277.554} C_VEL
LIN {X 0,Y 474.277,Z 596.501,A -85,B 0,C 180,E1 -7279.328,E2 -7279.328} C_VEL
LIN {X 0,Y 474.01,Z 602.47,A -85,B 0,C 180,E1 -7281.046,E2 -7281.046} C_VEL
LIN {X 0,Y 473.88,Z 608.25,A -85,B 0,C 180,E1 -7283.188,E2 -7283.188} C_VEL
LIN {X 0,Y 473.762,Z 611.637,A -85,B 0,C 180,E1 -7284.896,E2 -7284.896} C_VEL
LIN {X 0,Y 473.742,Z 614.093,A -85,B 0,C 180,E1 -7286.6,E2 -7286.6} C_VEL
LIN {X 0,Y 473.689,Z 615.48,A -85,B 0,C 180,E1 -7288.302,E2 -7288.302} C_VEL
LIN {X 0,Y 473.665,Z 616,A -85,B 0,C 180,E1 -7290.002,E2 -7290.002} C_VEL
LIN {X 0,Y 473.689,Z 615.477,A -85,B 0,C 180,E1 -7291.702,E2 -7291.702} C_VEL
LIN {X 0,Y 473.743,Z 614.087,A -85,B 0,C 180,E1 -7293.404,E2 -7293.404} C_VEL
LIN {X 0,Y 473.764,Z 611.63,A -85,B 0,C 180,E1 -7295.108,E2 -7295.108} C_VEL
LIN {X 0,Y 473.884,Z 608.247,A -85,B 0,C 180,E1 -7296.816,E2 -7296.816} C_VEL
LIN {X 0,Y 474.007,Z 602.462,A -85,B 0,C 180,E1 -7298.958,E2 -7298.958} C_VEL
LIN {X 0,Y 474.355,Z 594.848,A -85,B 0,C 180,E1 -7301.107,E2 -7301.107} C_VEL
LIN {X 0,Y 474.751,Z 587.258,A -85,B 0,C 180,E1 -7302.831,E2 -7302.831} C_VEL
LIN {X 0,Y 475.336,Z 578.197,A -85,B 0,C 180,E1 -7304.559,E2 -7304.559} C_VEL
LIN {X 0,Y 475.995,Z 568.895,A -85,B 0,C 180,E1 -7306.073,E2 -7306.073} C_VEL
LIN {X 0,Y 476.808,Z 557.991,A -85,B 0,C 180,E1 -7307.589,E2 -7307.589} C_VEL
LIN {X 0,Y 477.661,Z 547.048,A -85,B 0,C 180,E1 -7308.888,E2 -7308.888} C_VEL
LIN {X 0,Y 478.656,Z 534.779,A -85,B 0,C 180,E1 -7310.147,E2 -7310.147} C_VEL
LIN {X 0,Y 479.646,Z 522.003,A -85,B 0,C 180,E1 -7311.265,E2 -7311.265} C_VEL
LIN {X 0,Y 480.584,Z 508.842,A -85,B 0,C 180,E1 -7312.236,E2 -7312.236} C_VEL
LIN {X 0,Y 481.69,Z 493.041,A -85,B 0,C 180,E1 -7313.201,E2 -7313.201} C_VEL
LIN {X 0,Y 482.516,Z 477.8,A -85,B 0,C 180,E1 -7313.956,E2 -7313.956} C_VEL
LIN {X 0,Y 483.325,Z 461.004,A -85,B 0,C 180,E1 -7314.591,E2 -7314.591} C_VEL
LIN {X 0,Y 483.906,Z 444.719,A -85,B 0,C 180,E1 -7315.025,E2 -7315.025} C_VEL
LIN {X 0,Y 483.147,Z 439.993,A -85,B 0,C 180,E1 -7315.17,E2 -7315.17} C_VEL
LIN {X 0,Y 478.843,Z 420.478,A -85,B 0,C 180,E1 -7315.745,E2 -7315.745} C_VEL
LIN {X 0,Y 479.8,Z 398.939,A -85,B 0,C 180,E1 -7318.908,E2 -7318.908} C_VEL
LIN {X 0,Y 481.321,Z 376.254,A -85,B 0,C 180,E1 -7322.511,E2 -7322.511} C_VEL
LIN {X 0,Y 482.676,Z 361.513,A -85,B 0,C 180,E1 -7325.041,E2 -7325.041} C_VEL
LIN {X 0,Y 483.711,Z 353.426,A -85,B 0,C 180,E1 -7326.564,E2 -7326.564} C_VEL
LIN {X 0,Y 482.404,Z 347.056,A -85,B 0,C 180,E1 -7328.121,E2 -7328.121} C_VEL
LIN {X 0,Y 480.521,Z 340.58,A -85,B 0,C 180,E1 -7330.057,E2 -7330.057} C_VEL
LIN {X 0,Y 479.199,Z 336.443,A -85,B 0,C 180,E1 -7331.585,E2 -7331.585} C_VEL
LIN {X 0,Y 477.782,Z 332.147,A -85,B 0,C 180,E1 -7333.739,E2 -7333.739} C_VEL
LIN {X 0,Y 477.207,Z 330.419,A -85,B 0,C 180,E1 -7335.016,E2 -7335.016} C_VEL
LIN {X 0,Y 476.847,Z 329.326,A -85,B 0,C 180,E1 -7336.237,E2 -7336.237} C_VEL
LIN {X 0,Y 476.643,Z 328.758,A -85,B 0,C 180,E1 -7337.498,E2 -7337.498} C_VEL
LIN {X 0,Y 476.576,Z 329.069,A -85,B 0,C 180,E1 -7339.545,E2 -7339.545} C_VEL
LIN {X 0,Y 476.882,Z 330.729,A -85,B 0,C 180,E1 -7341.759,E2 -7341.759} C_VEL
LIN {X 0,Y 477.207,Z 333.66,A -85,B 0,C 180,E1 -7344.098,E2 -7344.098} C_VEL
LIN {X 0,Y 477.05,Z 336.605,A -85,B 0,C 180,E1 -7345.957,E2 -7345.957} C_VEL
LIN {X 0,Y 476.469,Z 341.779,A -85,B 0,C 180,E1 -7348.919,E2 -7348.919} C_VEL
LIN {X 0,Y 476.119,Z 346.961,A -85,B 0,C 180,E1 -7351.813,E2 -7351.813} C_VEL
LIN {X 0,Y 475.877,Z 352.03,A -85,B 0,C 180,E1 -7354.641,E2 -7354.641} C_VEL
LIN {X 0,Y 475.636,Z 357.034,A -85,B 0,C 180,E1 -7357.408,E2 -7357.408} C_VEL
LIN {X 0,Y 475.426,Z 361.954,A -85,B 0,C 180,E1 -7360.124,E2 -7360.124} C_VEL
LIN {X 0,Y 475.181,Z 368.46,A -85,B 0,C 180,E1 -7363.68,E2 -7363.68} C_VEL
LIN {X 0,Y 475.144,Z 369.402,A -85,B 0,C 180,E1 -7364.19,E2 -7364.19} C_VEL
LIN {X 0,Y 479.013,Z 381.833,A -85,B 0,C 180,E1 -7364.823,E2 -7364.823} C_VEL
LIN {X 0,Y 478.572,Z 395.451,A -85,B 0,C 180,E1 -7365.435,E2 -7365.435} C_VEL
LIN {X 0,Y 477.973,Z 407.696,A -85,B 0,C 180,E1 -7366.155,E2 -7366.155} C_VEL
LIN {X 0,Y 477.476,Z 419.547,A -85,B 0,C 180,E1 -7367.04,E2 -7367.04} C_VEL
LIN {X 0,Y 476.902,Z 430.88,A -85,B 0,C 180,E1 -7368.094,E2 -7368.094} C_VEL
LIN {X 0,Y 476.481,Z 440.193,A -85,B 0,C 180,E1 -7369.161,E2 -7369.161} C_VEL
LIN {X 0,Y 475.975,Z 449.342,A -85,B 0,C 180,E1 -7370.439,E2 -7370.439} C_VEL
LIN {X 0,Y 475.583,Z 456.825,A -85,B 0,C 180,E1 -7371.749,E2 -7371.749} C_VEL
LIN {X 0,Y 475.151,Z 463.412,A -85,B 0,C 180,E1 -7373.205,E2 -7373.205} C_VEL
LIN {X 0,Y 474.929,Z 467.872,A -85,B 0,C 180,E1 -7374.481,E2 -7374.481} C_VEL
LIN {X 0,Y 474.853,Z 471.243,A -85,B 0,C 180,E1 -7375.756,E2 -7375.756} C_VEL
LIN {X 0,Y 474.747,Z 472.965,A -85,B 0,C 180,E1 -7376.606,E2 -7376.606} C_VEL
LIN {X 0,Y 474.597,Z 474.258,A -85,B 0,C 180,E1 -7377.454,E2 -7377.454} C_VEL
LIN {X 0,Y 474.46,Z 475.128,A -85,B 0,C 180,E1 -7378.303,E2 -7378.303} C_VEL
LIN {X 0,Y 474.358,Z 475.675,A -85,B 0,C 180,E1 -7380,E2 -7380} C_VEL
LIN {X 0,Y 474.362,Z 475.35,A -85,B 0,C 180,E1 -7380.849,E2 -7380.849} C_VEL
LIN {X 0,Y 474.43,Z 474.597,A -85,B 0,C 180,E1 -7381.698,E2 -7381.698} C_VEL
LIN {X 0,Y 474.454,Z 473.467,A -85,B 0,C 180,E1 -7382.547,E2 -7382.547} C_VEL
LIN {X 0,Y 474.561,Z 471.916,A -85,B 0,C 180,E1 -7383.396,E2 -7383.396} C_VEL
LIN {X 0,Y 474.511,Z 468.811,A -85,B 0,C 180,E1 -7384.673,E2 -7384.673} C_VEL
LIN {X 0,Y 474.696,Z 464.648,A -85,B 0,C 180,E1 -7385.949,E2 -7385.949} C_VEL
LIN {X 0,Y 474.891,Z 458.309,A -85,B 0,C 180,E1 -7387.45,E2 -7387.45} C_VEL
LIN {X 0,Y 475.217,Z 450.213,A -85,B 0,C 180,E1 -7388.934,E2 -7388.934} C_VEL
LIN {X 0,Y 475.508,Z 441.467,A -85,B 0,C 180,E1 -7390.216,E2 -7390.216} C_VEL
LIN {X 0,Y 476.013,Z 431.516,A -85,B 0,C 180,E1 -7391.39,E2 -7391.39} C_VEL
LIN {X 0,Y 476.386,Z 420.409,A -85,B 0,C 180,E1 -7392.46,E2 -7392.46} C_VEL
LIN {X 0,Y 476.81,Z 408.316,A -85,B 0,C 180,E1 -7393.387,E2 -7393.387} C_VEL
LIN {X 0,Y 477.372,Z 395.241,A -85,B 0,C 180,E1 -7394.168,E2 -7394.168} C_VEL
LIN {X 0,Y 477.687,Z 382.195,A -85,B 0,C 180,E1 -7394.757,E2 -7394.757} C_VEL
LIN {X 0,Y 477.551,Z 378.25,A -85,B 0,C 180,E1 -7394.911,E2 -7394.911} C_VEL
LIN {X 0,Y 474.24,Z 364.375,A -85,B 0,C 180,E1 -7395.441,E2 -7395.441} C_VEL
LIN {X 0,Y 474.314,Z 358.2,A -85,B 0,C 180,E1 -7398.502,E2 -7398.502} C_VEL
LIN {X 0,Y 474.443,Z 351.713,A -85,B 0,C 180,E1 -7401.736,E2 -7401.736} C_VEL
LIN {X 0,Y 474.565,Z 346.234,A -85,B 0,C 180,E1 -7404.498,E2 -7404.498} C_VEL
LIN {X 0,Y 474.682,Z 340.674,A -85,B 0,C 180,E1 -7407.332,E2 -7407.332} C_VEL
LIN {X 0,Y 474.82,Z 335.076,A -85,B 0,C 180,E1 -7410.215,E2 -7410.215} C_VEL
LIN {X 0,Y 474.971,Z 329.338,A -85,B 0,C 180,E1 -7413.195,E2 -7413.195} C_VEL
LIN {X 0,Y 474.997,Z 324.886,A -85,B 0,C 180,E1 -7415.532,E2 -7415.532} C_VEL
LIN {X 0,Y 474.633,Z 321.68,A -85,B 0,C 180,E1 -7417.38,E2 -7417.38} C_VEL
LIN {X 0,Y 474.623,Z 321.679,A -85,B 0,C 180,E1 -7420.658,E2 -7420.658} C_VEL
LIN {X 0,Y 474.6,Z 321.68,A -85,B 0,C 180,E1 -7423.479,E2 -7423.479} C_VEL
LIN {X 0,Y 474.599,Z 321.681,A -85,B 0,C 180,E1 -7426.52,E2 -7426.52} C_VEL
LIN {X 0,Y 474.623,Z 321.678,A -85,B 0,C 180,E1 -7429.341,E2 -7429.341} C_VEL
LIN {X 0,Y 474.626,Z 321.68,A -85,B 0,C 180,E1 -7432.618,E2 -7432.618} C_VEL
LIN {X 0,Y 474.625,Z 321.788,A -85,B 0,C 180,E1 -7433.093,E2 -7433.093} C_VEL
LIN {X 0,Y 475.253,Z 325.876,A -85,B 0,C 180,E1 -7434.778,E2 -7434.778} C_VEL
LIN {X 0,Y 475.267,Z 330.703,A -85,B 0,C 180,E1 -7436.828,E2 -7436.828} C_VEL
LIN {X 0,Y 475.163,Z 337.277,A -85,B 0,C 180,E1 -7439.807,E2 -7439.807} C_VEL
LIN {X 0,Y 475.054,Z 343.234,A -85,B 0,C 180,E1 -7442.7,E2 -7442.7} C_VEL
LIN {X 0,Y 474.974,Z 346.687,A -85,B 0,C 180,E1 -7444.399,E2 -7444.399} C_VEL
LIN {X 0,Y 474.321,Z 348.205,A -85,B 0,C 180,E1 -7445.082,E2 -7445.082} C_VEL
LIN {X 0,Y 471.45,Z 350.976,A -85,B 0,C 180,E1 -7446.183,E2 -7446.183} C_VEL
LIN {X 0,Y 469.014,Z 353.23,A -85,B 0,C 180,E1 -7447.068,E2 -7447.068} C_VEL
LIN {X 0,Y 467.973,Z 354.84,A -85,B 0,C 180,E1 -7447.757,E2 -7447.757} C_VEL
LIN {X 0,Y 467.893,Z 355.345,A -85,B 0,C 180,E1 -7447.991,E2 -7447.991} C_VEL
LIN {X 0,Y 467.881,Z 362.218,A -85,B 0,C 180,E1 -7451.142,E2 -7451.142} C_VEL
LIN {X 0,Y 467.943,Z 369.844,A -85,B 0,C 180,E1 -7454.314,E2 -7454.314} C_VEL
LIN {X 0,Y 467.991,Z 370.762,A -85,B 0,C 180,E1 -7454.678,E2 -7454.678} C_VEL
LIN {X 0,Y 470.889,Z 381.432,A -85,B 0,C 180,E1 -7455.051,E2 -7455.051} C_VEL
LIN {X 0,Y 470.673,Z 393.873,A -85,B 0,C 180,E1 -7455.514,E2 -7455.514} C_VEL
LIN {X 0,Y 470.36,Z 406.439,A -85,B 0,C 180,E1 -7456.167,E2 -7456.167} C_VEL
LIN {X 0,Y 470.107,Z 417.344,A -85,B 0,C 180,E1 -7456.915,E2 -7456.915} C_VEL
LIN {X 0,Y 469.691,Z 427.573,A -85,B 0,C 180,E1 -7457.797,E2 -7457.797} C_VEL
LIN {X 0,Y 469.222,Z 436.797,A -85,B 0,C 180,E1 -7458.77,E2 -7458.77} C_VEL
LIN {X 0,Y 468.866,Z 445.2,A -85,B 0,C 180,E1 -7459.854,E2 -7459.854} C_VEL
LIN {X 0,Y 468.431,Z 452.147,A -85,B 0,C 180,E1 -7460.934,E2 -7460.934} C_VEL
LIN {X 0,Y 468.185,Z 458.935,A -85,B 0,C 180,E1 -7462.234,E2 -7462.234} C_VEL
LIN {X 0,Y 467.91,Z 464.336,A -85,B 0,C 180,E1 -7463.53,E2 -7463.53} C_VEL
LIN {X 0,Y 467.557,Z 468.594,A -85,B 0,C 180,E1 -7464.824,E2 -7464.824} C_VEL
LIN {X 0,Y 467.509,Z 470.812,A -85,B 0,C 180,E1 -7465.687,E2 -7465.687} C_VEL
LIN {X 0,Y 467.489,Z 472.618,A -85,B 0,C 180,E1 -7466.55,E2 -7466.55} C_VEL
LIN {X 0,Y 467.408,Z 474.01,A -85,B 0,C 180,E1 -7467.413,E2 -7467.413} C_VEL
LIN {X 0,Y 467.335,Z 475.584,A -85,B 0,C 180,E1 -7469.136,E2 -7469.136} C_VEL
LIN {X 0,Y 467.317,Z 475.819,A -85,B 0,C 180,E1 -7469.998,E2 -7469.998} C_VEL
LIN {X 0,Y 467.334,Z 475.635,A -85,B 0,C 180,E1 -7470.86,E2 -7470.86} C_VEL
LIN {X 0,Y 467.423,Z 474.124,A -85,B 0,C 180,E1 -7472.583,E2 -7472.583} C_VEL
LIN {X 0,Y 467.567,Z 472.787,A -85,B 0,C 180,E1 -7473.445,E2 -7473.445} C_VEL
LIN {X 0,Y 467.637,Z 470.004,A -85,B 0,C 180,E1 -7474.739,E2 -7474.739} C_VEL
LIN {X 0,Y 467.787,Z 466.211,A -85,B 0,C 180,E1 -7476.035,E2 -7476.035} C_VEL
LIN {X 0,Y 467.986,Z 461.509,A -85,B 0,C 180,E1 -7477.281,E2 -7477.281} C_VEL
LIN {X 0,Y 468.333,Z 455.068,A -85,B 0,C 180,E1 -7478.628,E2 -7478.628} C_VEL
LIN {X 0,Y 468.753,Z 447.321,A -85,B 0,C 180,E1 -7479.926,E2 -7479.926} C_VEL
LIN {X 0,Y 469.114,Z 439.405,A -85,B 0,C 180,E1 -7481.01,E2 -7481.01} C_VEL
LIN {X 0,Y 469.553,Z 429.679,A -85,B 0,C 180,E1 -7482.093,E2 -7482.093} C_VEL
LIN {X 0,Y 469.918,Z 420.067,A -85,B 0,C 180,E1 -7482.961,E2 -7482.961} C_VEL
LIN {X 0,Y 470.286,Z 407.979,A -85,B 0,C 180,E1 -7483.831,E2 -7483.831} C_VEL
LIN {X 0,Y 470.659,Z 395.971,A -85,B 0,C 180,E1 -7484.482,E2 -7484.482} C_VEL
LIN {X 0,Y 470.884,Z 382.652,A -85,B 0,C 180,E1 -7485,E2 -7485} C_VEL
LIN {X 0,Y 470.527,Z 379.667,A -85,B 0,C 180,E1 -7485.103,E2 -7485.103} C_VEL
LIN {X 0,Y 467.981,Z 370.747,A -85,B 0,C 180,E1 -7485.43,E2 -7485.43} C_VEL
LIN {X 0,Y 467.86,Z 363.523,A -85,B 0,C 180,E1 -7488.386,E2 -7488.386} C_VEL
LIN {X 0,Y 467.917,Z 356.896,A -85,B 0,C 180,E1 -7491.372,E2 -7491.372} C_VEL
LIN {X 0,Y 467.937,Z 351.588,A -85,B 0,C 180,E1 -7493.921,E2 -7493.921} C_VEL
LIN {X 0,Y 468.048,Z 345.829,A -85,B 0,C 180,E1 -7496.771,E2 -7496.771} C_VEL
LIN {X 0,Y 468.245,Z 338.794,A -85,B 0,C 180,E1 -7500.183,E2 -7500.183} C_VEL
LIN {X 0,Y 468.321,Z 332.119,A -85,B 0,C 180,E1 -7503.22,E2 -7503.22} C_VEL
LIN {X 0,Y 468.281,Z 327.312,A -85,B 0,C 180,E1 -7505.293,E2 -7505.293} C_VEL
LIN {X 0,Y 467.58,Z 322.557,A -85,B 0,C 180,E1 -7507.263,E2 -7507.263} C_VEL
LIN {X 0,Y 467.557,Z 322.559,A -85,B 0,C 180,E1 -7510.263,E2 -7510.263} C_VEL
LIN {X 0,Y 467.536,Z 322.561,A -85,B 0,C 180,E1 -7513.743,E2 -7513.743} C_VEL
LIN {X 0,Y 467.562,Z 322.554,A -85,B 0,C 180,E1 -7516.256,E2 -7516.256} C_VEL
LIN {X 0,Y 467.575,Z 322.558,A -85,B 0,C 180,E1 -7518.719,E2 -7518.719} C_VEL
LIN {X 0,Y 467.564,Z 322.554,A -85,B 0,C 180,E1 -7521.404,E2 -7521.404} C_VEL
LIN {X 0,Y 467.544,Z 322.558,A -85,B 0,C 180,E1 -7524.258,E2 -7524.258} C_VEL
LIN {X 0,Y 467.562,Z 322.556,A -85,B 0,C 180,E1 -7527.319,E2 -7527.319} C_VEL
LIN {X 0,Y 467.549,Z 322.556,A -85,B 0,C 180,E1 -7530.666,E2 -7530.666} C_VEL
LIN {X 0,Y 467.607,Z 322.545,A -85,B 0,C 180,E1 -7533.199,E2 -7533.199} C_VEL
LIN {X 0,Y 467.568,Z 322.557,A -85,B 0,C 180,E1 -7536.056,E2 -7536.056} C_VEL
LIN {X 0,Y 467.619,Z 322.547,A -85,B 0,C 180,E1 -7538.856,E2 -7538.856} C_VEL
LIN {X 0,Y 467.608,Z 322.548,A -85,B 0,C 180,E1 -7541.601,E2 -7541.601} C_VEL
LIN {X 0,Y 467.614,Z 322.548,A -85,B 0,C 180,E1 -7544.304,E2 -7544.304} C_VEL
LIN {X 0,Y 467.677,Z 322.54,A -85,B 0,C 180,E1 -7547.855,E2 -7547.855} C_VEL
LIN {X 0,Y 467.665,Z 322.537,A -85,B 0,C 180,E1 -7551.357,E2 -7551.357} C_VEL
LIN {X 0,Y 467.723,Z 322.534,A -85,B 0,C 180,E1 -7553.962,E2 -7553.962} C_VEL
LIN {X 0,Y 467.831,Z 322.523,A -85,B 0,C 180,E1 -7557.417,E2 -7557.417} C_VEL
LIN {X 0,Y 467.854,Z 322.515,A -85,B 0,C 180,E1 -7560,E2 -7560} C_VEL
LIN {X 0,Y 467.845,Z 322.522,A -85,B 0,C 180,E1 -7562.583,E2 -7562.583} C_VEL
LIN {X 0,Y 467.731,Z 322.536,A -85,B 0,C 180,E1 -7566.037,E2 -7566.037} C_VEL
LIN {X 0,Y 467.659,Z 322.542,A -85,B 0,C 180,E1 -7568.643,E2 -7568.643} C_VEL
LIN {X 0,Y 467.658,Z 322.543,A -85,B 0,C 180,E1 -7572.145,E2 -7572.145} C_VEL
LIN {X 0,Y 467.642,Z 322.546,A -85,B 0,C 180,E1 -7575.894,E2 -7575.894} C_VEL
LIN {X 0,Y 467.601,Z 322.55,A -85,B 0,C 180,E1 -7579.308,E2 -7579.308} C_VEL
LIN {X 0,Y 467.554,Z 322.556,A -85,B 0,C 180,E1 -7582.073,E2 -7582.073} C_VEL
LIN {X 0,Y 467.584,Z 322.555,A -85,B 0,C 180,E1 -7584.888,E2 -7584.888} C_VEL
LIN {X 0,Y 467.596,Z 322.549,A -85,B 0,C 180,E1 -7587.77,E2 -7587.77} C_VEL
LIN {X 0,Y 467.546,Z 322.557,A -85,B 0,C 180,E1 -7591.047,E2 -7591.047} C_VEL
LIN {X 0,Y 467.568,Z 322.556,A -85,B 0,C 180,E1 -7594.244,E2 -7594.244} C_VEL
LIN {X 0,Y 467.531,Z 322.562,A -85,B 0,C 180,E1 -7597.189,E2 -7597.189} C_VEL
LIN {X 0,Y 467.557,Z 322.556,A -85,B 0,C 180,E1 -7600.266,E2 -7600.266} C_VEL
LIN {X 0,Y 467.567,Z 322.557,A -85,B 0,C 180,E1 -7602.569,E2 -7602.569} C_VEL
LIN {X 0,Y 467.591,Z 322.653,A -85,B 0,C 180,E1 -7605.686,E2 -7605.686} C_VEL
LIN {X 0,Y 471.033,Z 333.899,A -85,B 0,C 180,E1 -7608.527,E2 -7608.527} C_VEL
LIN {X 0,Y 474.571,Z 345.93,A -85,B 0,C 180,E1 -7611.327,E2 -7611.327} C_VEL
LIN {X 0,Y 476.604,Z 353.929,A -85,B 0,C 180,E1 -7613.038,E2 -7613.038} C_VEL
LIN {X 0,Y 476.73,Z 356.957,A -85,B 0,C 180,E1 -7613.607,E2 -7613.607} C_VEL
LIN {X 0,Y 475.092,Z 374.174,A -85,B 0,C 180,E1 -7616.565,E2 -7616.565} C_VEL
LIN {X 0,Y 473.646,Z 393.287,A -85,B 0,C 180,E1 -7619.705,E2 -7619.705} C_VEL
LIN {X 0,Y 472.403,Z 412.713,A -85,B 0,C 180,E1 -7622.752,E2 -7622.752} C_VEL
LIN {X 0,Y 471.996,Z 420.384,A -85,B 0,C 180,E1 -7623.926,E2 -7623.926} C_VEL
LIN {X 0,Y 477.422,Z 444.777,A -85,B 0,C 180,E1 -7624.638,E2 -7624.638} C_VEL
LIN {X 0,Y 476.752,Z 461.771,A -85,B 0,C 180,E1 -7625.092,E2 -7625.092} C_VEL
LIN {X 0,Y 476.005,Z 477.813,A -85,B 0,C 180,E1 -7625.7,E2 -7625.7} C_VEL
LIN {X 0,Y 475.091,Z 493.123,A -85,B 0,C 180,E1 -7626.462,E2 -7626.462} C_VEL
LIN {X 0,Y 473.984,Z 508.906,A -85,B 0,C 180,E1 -7627.442,E2 -7627.442} C_VEL
LIN {X 0,Y 472.858,Z 523.346,A -85,B 0,C 180,E1 -7628.534,E2 -7628.534} C_VEL
LIN {X 0,Y 471.781,Z 536.731,A -85,B 0,C 180,E1 -7629.739,E2 -7629.739} C_VEL
LIN {X 0,Y 470.707,Z 549.032,A -85,B 0,C 180,E1 -7631.053,E2 -7631.053} C_VEL
LIN {X 0,Y 469.677,Z 561.277,A -85,B 0,C 180,E1 -7632.589,E2 -7632.589} C_VEL
LIN {X 0,Y 468.947,Z 571.825,A -85,B 0,C 180,E1 -7634.148,E2 -7634.148} C_VEL
LIN {X 0,Y 468.096,Z 581.834,A -85,B 0,C 180,E1 -7635.881,E2 -7635.881} C_VEL
LIN {X 0,Y 467.586,Z 590.497,A -85,B 0,C 180,E1 -7637.679,E2 -7637.679} C_VEL
LIN {X 0,Y 467.234,Z 596.5,A -85,B 0,C 180,E1 -7639.165,E2 -7639.165} C_VEL
LIN {X 0,Y 466.941,Z 602.469,A -85,B 0,C 180,E1 -7640.909,E2 -7640.909} C_VEL
LIN {X 0,Y 466.811,Z 608.25,A -85,B 0,C 180,E1 -7643.085,E2 -7643.085} C_VEL
LIN {X 0,Y 466.669,Z 611.637,A -85,B 0,C 180,E1 -7644.818,E2 -7644.818} C_VEL
LIN {X 0,Y 466.637,Z 614.093,A -85,B 0,C 180,E1 -7646.548,E2 -7646.548} C_VEL
LIN {X 0,Y 466.598,Z 615.479,A -85,B 0,C 180,E1 -7648.276,E2 -7648.276} C_VEL
LIN {X 0,Y 466.565,Z 616,A -85,B 0,C 180,E1 -7650.002,E2 -7650.002} C_VEL
LIN {X 0,Y 466.598,Z 615.476,A -85,B 0,C 180,E1 -7651.728,E2 -7651.728} C_VEL
LIN {X 0,Y 466.638,Z 614.087,A -85,B 0,C 180,E1 -7653.456,E2 -7653.456} C_VEL
LIN {X 0,Y 466.671,Z 611.63,A -85,B 0,C 180,E1 -7655.186,E2 -7655.186} C_VEL
LIN {X 0,Y 466.815,Z 608.247,A -85,B 0,C 180,E1 -7656.92,E2 -7656.92} C_VEL
LIN {X 0,Y 466.939,Z 602.461,A -85,B 0,C 180,E1 -7659.095,E2 -7659.095} C_VEL
LIN {X 0,Y 467.307,Z 594.848,A -85,B 0,C 180,E1 -7661.276,E2 -7661.276} C_VEL
LIN {X 0,Y 467.733,Z 587.258,A -85,B 0,C 180,E1 -7663.027,E2 -7663.027} C_VEL
LIN {X 0,Y 468.36,Z 578.197,A -85,B 0,C 180,E1 -7664.781,E2 -7664.781} C_VEL
LIN {X 0,Y 469.093,Z 568.623,A -85,B 0,C 180,E1 -7666.357,E2 -7666.357} C_VEL
LIN {X 0,Y 469.953,Z 557.991,A -85,B 0,C 180,E1 -7667.854,E2 -7667.854} C_VEL
LIN {X 0,Y 470.865,Z 547.047,A -85,B 0,C 180,E1 -7669.171,E2 -7669.171} C_VEL
LIN {X 0,Y 471.933,Z 534.833,A -85,B 0,C 180,E1 -7670.441,E2 -7670.441} C_VEL
LIN {X 0,Y 472.995,Z 522.001,A -85,B 0,C 180,E1 -7671.579,E2 -7671.579} C_VEL
LIN {X 0,Y 473.989,Z 508.841,A -85,B 0,C 180,E1 -7672.562,E2 -7672.562} C_VEL
LIN {X 0,Y 475.125,Z 493.039,A -85,B 0,C 180,E1 -7673.541,E2 -7673.541} C_VEL
LIN {X 0,Y 476.019,Z 477.714,A -85,B 0,C 180,E1 -7674.304,E2 -7674.304} C_VEL
LIN {X 0,Y 476.777,Z 461.819,A -85,B 0,C 180,E1 -7674.904,E2 -7674.904} C_VEL
LIN {X 0,Y 477.347,Z 445.778,A -85,B 0,C 180,E1 -7675.335,E2 -7675.335} C_VEL
LIN {X 0,Y 475.142,Z 434.648,A -85,B 0,C 180,E1 -7675.659,E2 -7675.659} C_VEL
LIN {X 0,Y 471.97,Z 420.156,A -85,B 0,C 180,E1 -7676.06,E2 -7676.06} C_VEL
LIN {X 0,Y 473.054,Z 398.197,A -85,B 0,C 180,E1 -7679.36,E2 -7679.36} C_VEL
LIN {X 0,Y 474.603,Z 377.591,A -85,B 0,C 180,E1 -7682.727,E2 -7682.727} C_VEL
LIN {X 0,Y 475.988,Z 363.776,A -85,B 0,C 180,E1 -7685.16,E2 -7685.16} C_VEL
LIN {X 0,Y 477.069,Z 356.18,A -85,B 0,C 180,E1 -7686.631,E2 -7686.631} C_VEL
LIN {X 0,Y 476.051,Z 350.403,A -85,B 0,C 180,E1 -7688.052,E2 -7688.052} C_VEL
LIN {X 0,Y 474.559,Z 345.016,A -85,B 0,C 180,E1 -7689.638,E2 -7689.638} C_VEL
LIN {X 0,Y 473.06,Z 340.18,A -85,B 0,C 180,E1 -7691.388,E2 -7691.388} C_VEL
LIN {X 0,Y 471.709,Z 336.221,A -85,B 0,C 180,E1 -7693.265,E2 -7693.265} C_VEL
LIN {X 0,Y 471.076,Z 334.253,A -85,B 0,C 180,E1 -7694.525,E2 -7694.525} C_VEL
LIN {X 0,Y 470.398,Z 332.258,A -85,B 0,C 180,E1 -7696.586,E2 -7696.586} C_VEL
LIN {X 0,Y 470.154,Z 331.75,A -85,B 0,C 180,E1 -7698.369,E2 -7698.369} C_VEL
LIN {X 0,Y 470.151,Z 332.156,A -85,B 0,C 180,E1 -7700.001,E2 -7700.001} C_VEL
LIN {X 0,Y 470.357,Z 334.043,A -85,B 0,C 180,E1 -7702.367,E2 -7702.367} C_VEL
LIN {X 0,Y 470.495,Z 336.473,A -85,B 0,C 180,E1 -7704.369,E2 -7704.369} C_VEL
LIN {X 0,Y 470.167,Z 339.629,A -85,B 0,C 180,E1 -7706.422,E2 -7706.422} C_VEL
LIN {X 0,Y 469.487,Z 346.345,A -85,B 0,C 180,E1 -7710.397,E2 -7710.397} C_VEL
LIN {X 0,Y 469.098,Z 351.425,A -85,B 0,C 180,E1 -7713.291,E2 -7713.291} C_VEL
LIN {X 0,Y 468.832,Z 356.426,A -85,B 0,C 180,E1 -7716.125,E2 -7716.125} C_VEL
LIN {X 0,Y 468.617,Z 361.391,A -85,B 0,C 180,E1 -7718.904,E2 -7718.904} C_VEL
LIN {X 0,Y 468.367,Z 366.292,A -85,B 0,C 180,E1 -7721.633,E2 -7721.633} C_VEL
LIN {X 0,Y 468.247,Z 370.443,A -85,B 0,C 180,E1 -7723.863,E2 -7723.863} C_VEL
LIN {X 0,Y 472.336,Z 382.772,A -85,B 0,C 180,E1 -7724.521,E2 -7724.521} C_VEL
LIN {X 0,Y 471.98,Z 395.674,A -85,B 0,C 180,E1 -7725.116,E2 -7725.116} C_VEL
LIN {X 0,Y 471.314,Z 408.637,A -85,B 0,C 180,E1 -7725.888,E2 -7725.888} C_VEL
LIN {X 0,Y 470.733,Z 421.156,A -85,B 0,C 180,E1 -7726.84,E2 -7726.84} C_VEL
LIN {X 0,Y 470.119,Z 432.449,A -85,B 0,C 180,E1 -7727.919,E2 -7727.919} C_VEL
LIN {X 0,Y 469.669,Z 441.657,A -85,B 0,C 180,E1 -7729.002,E2 -7729.002} C_VEL
LIN {X 0,Y 469.11,Z 450.738,A -85,B 0,C 180,E1 -7730.297,E2 -7730.297} C_VEL
LIN {X 0,Y 468.696,Z 458.057,A -85,B 0,C 180,E1 -7731.601,E2 -7731.601} C_VEL
LIN {X 0,Y 468.229,Z 464.751,A -85,B 0,C 180,E1 -7733.104,E2 -7733.104} C_VEL
LIN {X 0,Y 467.983,Z 469.188,A -85,B 0,C 180,E1 -7734.399,E2 -7734.399} C_VEL
LIN {X 0,Y 467.903,Z 472.524,A -85,B 0,C 180,E1 -7735.693,E2 -7735.693} C_VEL
LIN {X 0,Y 467.774,Z 474.228,A -85,B 0,C 180,E1 -7736.555,E2 -7736.555} C_VEL
LIN {X 0,Y 467.615,Z 475.502,A -85,B 0,C 180,E1 -7737.416,E2 -7737.416} C_VEL
LIN {X 0,Y 467.469,Z 476.349,A -85,B 0,C 180,E1 -7738.277,E2 -7738.277} C_VEL
LIN {X 0,Y 467.38,Z 476.859,A -85,B 0,C 180,E1 -7740,E2 -7740} C_VEL
LIN {X 0,Y 467.361,Z 476.52,A -85,B 0,C 180,E1 -7740.862,E2 -7740.862} C_VEL
LIN {X 0,Y 467.427,Z 475.745,A -85,B 0,C 180,E1 -7741.724,E2 -7741.724} C_VEL
LIN {X 0,Y 467.565,Z 473.008,A -85,B 0,C 180,E1 -7743.447,E2 -7743.447} C_VEL
LIN {X 0,Y 467.51,Z 469.86,A -85,B 0,C 180,E1 -7744.743,E2 -7744.743} C_VEL
LIN {X 0,Y 467.723,Z 465.648,A -85,B 0,C 180,E1 -7746.038,E2 -7746.038} C_VEL
LIN {X 0,Y 467.925,Z 459.254,A -85,B 0,C 180,E1 -7747.563,E2 -7747.563} C_VEL
LIN {X 0,Y 468.241,Z 452.394,A -85,B 0,C 180,E1 -7748.85,E2 -7748.85} C_VEL
LIN {X 0,Y 468.542,Z 443.883,A -85,B 0,C 180,E1 -7750.152,E2 -7750.152} C_VEL
LIN {X 0,Y 468.933,Z 435.249,A -85,B 0,C 180,E1 -7751.235,E2 -7751.235} C_VEL
LIN {X 0,Y 469.377,Z 424.765,A -85,B 0,C 180,E1 -7752.32,E2 -7752.32} C_VEL
LIN {X 0,Y 469.845,Z 413.001,A -85,B 0,C 180,E1 -7753.301,E2 -7753.301} C_VEL
LIN {X 0,Y 470.342,Z 401.739,A -85,B 0,C 180,E1 -7754.053,E2 -7754.053} C_VEL
LIN {X 0,Y 470.698,Z 389.451,A -85,B 0,C 180,E1 -7754.704,E2 -7754.704} C_VEL
LIN {X 0,Y 470.77,Z 379.673,A -85,B 0,C 180,E1 -7755.11,E2 -7755.11} C_VEL
LIN {X 0,Y 467.516,Z 366.262,A -85,B 0,C 180,E1 -7755.641,E2 -7755.641} C_VEL
LIN {X 0,Y 467.203,Z 364.726,A -85,B 0,C 180,E1 -7755.71,E2 -7755.71} C_VEL
LIN {X 0,Y 467.282,Z 358.834,A -85,B 0,C 180,E1 -7758.64,E2 -7758.64} C_VEL
LIN {X 0,Y 467.412,Z 351.985,A -85,B 0,C 180,E1 -7762.08,E2 -7762.08} C_VEL
LIN {X 0,Y 467.535,Z 346.478,A -85,B 0,C 180,E1 -7764.892,E2 -7764.892} C_VEL
LIN {X 0,Y 467.685,Z 340.862,A -85,B 0,C 180,E1 -7767.765,E2 -7767.765} C_VEL
LIN {X 0,Y 467.826,Z 335.179,A -85,B 0,C 180,E1 -7770.716,E2 -7770.716} C_VEL
LIN {X 0,Y 467.983,Z 329.391,A -85,B 0,C 180,E1 -7773.756,E2 -7773.756} C_VEL
LIN {X 0,Y 467.936,Z 325.447,A -85,B 0,C 180,E1 -7775.856,E2 -7775.856} C_VEL
LIN {X 0,Y 467.596,Z 322.556,A -85,B 0,C 180,E1 -7777.468,E2 -7777.468} C_VEL
LIN {X 0,Y 467.578,Z 322.558,A -85,B 0,C 180,E1 -7780.265,E2 -7780.265} C_VEL
LIN {X 0,Y 467.569,Z 322.557,A -85,B 0,C 180,E1 -7782.563,E2 -7782.563} C_VEL
LIN {X 0,Y 467.574,Z 322.555,A -85,B 0,C 180,E1 -7785.052,E2 -7785.052} C_VEL
LIN {X 0,Y 467.582,Z 322.555,A -85,B 0,C 180,E1 -7788.596,E2 -7788.596} C_VEL
LIN {X 0,Y 467.579,Z 322.558,A -85,B 0,C 180,E1 -7791.955,E2 -7791.955} C_VEL
LIN {X 0,Y 467.611,Z 322.633,A -85,B 0,C 180,E1 -7792.882,E2 -7792.882} C_VEL
LIN {X 0,Y 468.345,Z 328.33,A -85,B 0,C 180,E1 -7795.232,E2 -7795.232} C_VEL
LIN {X 0,Y 468.247,Z 334.131,A -85,B 0,C 180,E1 -7797.802,E2 -7797.802} C_VEL
LIN {X 0,Y 468.127,Z 340.092,A -85,B 0,C 180,E1 -7800.547,E2 -7800.547} C_VEL
LIN {X 0,Y 468.022,Z 345.583,A -85,B 0,C 180,E1 -7803.223,E2 -7803.223} C_VEL
LIN {X 0,Y 467.952,Z 351.978,A -85,B 0,C 180,E1 -7806.368,E2 -7806.368} C_VEL
LIN {X 0,Y 467.893,Z 355.345,A -85,B 0,C 180,E1 -7807.991,E2 -7807.991} C_VEL
LIN {X 0,Y 467.238,Z 356.945,A -85,B 0,C 180,E1 -7808.683,E2 -7808.683} C_VEL
LIN {X 0,Y 464.399,Z 359.932,A -85,B 0,C 180,E1 -7809.793,E2 -7809.793} C_VEL
LIN {X 0,Y 462.001,Z 362.407,A -85,B 0,C 180,E1 -7810.685,E2 -7810.685} C_VEL
LIN {X 0,Y 460.989,Z 364.198,A -85,B 0,C 180,E1 -7811.378,E2 -7811.378} C_VEL
LIN {X 0,Y 460.916,Z 364.764,A -85,B 0,C 180,E1 -7811.614,E2 -7811.614} C_VEL
LIN {X 0,Y 461.054,Z 371.734,A -85,B 0,C 180,E1 -7814.442,E2 -7814.442} C_VEL
LIN {X 0,Y 464.092,Z 382.47,A -85,B 0,C 180,E1 -7814.827,E2 -7814.827} C_VEL
LIN {X 0,Y 463.863,Z 394.929,A -85,B 0,C 180,E1 -7815.297,E2 -7815.297} C_VEL
LIN {X 0,Y 463.539,Z 407.502,A -85,B 0,C 180,E1 -7815.959,E2 -7815.959} C_VEL
LIN {X 0,Y 463.278,Z 418.4,A -85,B 0,C 180,E1 -7816.718,E2 -7816.718} C_VEL
LIN {X 0,Y 462.839,Z 428.643,A -85,B 0,C 180,E1 -7817.613,E2 -7817.613} C_VEL
LIN {X 0,Y 462.34,Z 437.87,A -85,B 0,C 180,E1 -7818.601,E2 -7818.601} C_VEL
LIN {X 0,Y 461.984,Z 446.27,A -85,B 0,C 180,E1 -7819.701,E2 -7819.701} C_VEL
LIN {X 0,Y 461.509,Z 453.221,A -85,B 0,C 180,E1 -7820.797,E2 -7820.797} C_VEL
LIN {X 0,Y 461.231,Z 460.012,A -85,B 0,C 180,E1 -7822.116,E2 -7822.116} C_VEL
LIN {X 0,Y 460.946,Z 465.412,A -85,B 0,C 180,E1 -7823.432,E2 -7823.432} C_VEL
LIN {X 0,Y 460.567,Z 469.671,A -85,B 0,C 180,E1 -7824.745,E2 -7824.745} C_VEL
LIN {X 0,Y 460.511,Z 471.889,A -85,B 0,C 180,E1 -7825.622,E2 -7825.622} C_VEL
LIN {X 0,Y 460.502,Z 473.693,A -85,B 0,C 180,E1 -7826.498,E2 -7826.498} C_VEL
LIN {X 0,Y 460.402,Z 475.087,A -85,B 0,C 180,E1 -7827.373,E2 -7827.373} C_VEL
LIN {X 0,Y 460.325,Z 476.661,A -85,B 0,C 180,E1 -7829.123,E2 -7829.123} C_VEL
LIN {X 0,Y 460.305,Z 476.895,A -85,B 0,C 180,E1 -7829.998,E2 -7829.998} C_VEL
LIN {X 0,Y 460.323,Z 476.711,A -85,B 0,C 180,E1 -7830.873,E2 -7830.873} C_VEL
LIN {X 0,Y 460.418,Z 475.199,A -85,B 0,C 180,E1 -7832.622,E2 -7832.622} C_VEL
LIN {X 0,Y 460.569,Z 473.861,A -85,B 0,C 180,E1 -7833.497,E2 -7833.497} C_VEL
LIN {X 0,Y 460.644,Z 471.078,A -85,B 0,C 180,E1 -7834.811,E2 -7834.811} C_VEL
LIN {X 0,Y 460.814,Z 467.284,A -85,B 0,C 180,E1 -7836.126,E2 -7836.126} C_VEL
LIN {X 0,Y 461.103,Z 461.445,A -85,B 0,C 180,E1 -7837.651,E2 -7837.651} C_VEL
LIN {X 0,Y 461.468,Z 454.961,A -85,B 0,C 180,E1 -7838.978,E2 -7838.978} C_VEL
LIN {X 0,Y 461.917,Z 446.949,A -85,B 0,C 180,E1 -7840.296,E2 -7840.296} C_VEL
LIN {X 0,Y 462.314,Z 438.682,A -85,B 0,C 180,E1 -7841.396,E2 -7841.396} C_VEL
LIN {X 0,Y 462.782,Z 428.504,A -85,B 0,C 180,E1 -7842.496,E2 -7842.496} C_VEL
LIN {X 0,Y 463.283,Z 418.073,A -85,B 0,C 180,E1 -7843.4,E2 -7843.4} C_VEL
LIN {X 0,Y 463.549,Z 407.239,A -85,B 0,C 180,E1 -7844.148,E2 -7844.148} C_VEL
LIN {X 0,Y 463.913,Z 394.578,A -85,B 0,C 180,E1 -7844.809,E2 -7844.809} C_VEL
LIN {X 0,Y 463.976,Z 381.955,A -85,B 0,C 180,E1 -7845.285,E2 -7845.285} C_VEL
LIN {X 0,Y 461.021,Z 371.702,A -85,B 0,C 180,E1 -7845.668,E2 -7845.668} C_VEL
LIN {X 0,Y 460.906,Z 364.331,A -85,B 0,C 180,E1 -7848.673,E2 -7848.673} C_VEL
LIN {X 0,Y 460.945,Z 357.916,A -85,B 0,C 180,E1 -7851.554,E2 -7851.554} C_VEL
LIN {X 0,Y 460.959,Z 352.153,A -85,B 0,C 180,E1 -7854.306,E2 -7854.306} C_VEL
LIN {X 0,Y 461.087,Z 346.242,A -85,B 0,C 180,E1 -7857.208,E2 -7857.208} C_VEL
LIN {X 0,Y 461.272,Z 340.062,A -85,B 0,C 180,E1 -7860.182,E2 -7860.182} C_VEL
LIN {X 0,Y 461.349,Z 333.39,A -85,B 0,C 180,E1 -7863.255,E2 -7863.255} C_VEL
LIN {X 0,Y 461.313,Z 328.48,A -85,B 0,C 180,E1 -7865.371,E2 -7865.371} C_VEL
LIN {X 0,Y 460.538,Z 323.435,A -85,B 0,C 180,E1 -7867.482,E2 -7867.482} C_VEL
LIN {X 0,Y 460.522,Z 323.436,A -85,B 0,C 180,E1 -7870.266,E2 -7870.266} C_VEL
LIN {X 0,Y 460.495,Z 323.439,A -85,B 0,C 180,E1 -7873.372,E2 -7873.372} C_VEL
LIN {X 0,Y 460.51,Z 323.435,A -85,B 0,C 180,E1 -7876.625,E2 -7876.625} C_VEL
LIN {X 0,Y 460.548,Z 323.428,A -85,B 0,C 180,E1 -7879.725,E2 -7879.725} C_VEL
LIN {X 0,Y 460.512,Z 323.435,A -85,B 0,C 180,E1 -7882.517,E2 -7882.517} C_VEL
LIN {X 0,Y 460.529,Z 323.436,A -85,B 0,C 180,E1 -7885.622,E2 -7885.622} C_VEL
LIN {X 0,Y 460.517,Z 323.434,A -85,B 0,C 180,E1 -7888.743,E2 -7888.743} C_VEL
LIN {X 0,Y 460.568,Z 323.428,A -85,B 0,C 180,E1 -7892.25,E2 -7892.25} C_VEL
LIN {X 0,Y 460.563,Z 323.429,A -85,B 0,C 180,E1 -7894.705,E2 -7894.705} C_VEL
LIN {X 0,Y 460.519,Z 323.429,A -85,B 0,C 180,E1 -7897.571,E2 -7897.571} C_VEL
LIN {X 0,Y 460.547,Z 323.426,A -85,B 0,C 180,E1 -7900.383,E2 -7900.383} C_VEL
LIN {X 0,Y 460.541,Z 323.434,A -85,B 0,C 180,E1 -7903.145,E2 -7903.145} C_VEL
LIN {X 0,Y 460.535,Z 323.422,A -85,B 0,C 180,E1 -7905.867,E2 -7905.867} C_VEL
LIN {X 0,Y 460.618,Z 323.422,A -85,B 0,C 180,E1 -7908.559,E2 -7908.559} C_VEL
LIN {X 0,Y 460.671,Z 323.416,A -85,B 0,C 180,E1 -7912.108,E2 -7912.108} C_VEL
LIN {X 0,Y 460.676,Z 323.41,A -85,B 0,C 180,E1 -7914.748,E2 -7914.748} C_VEL
LIN {X 0,Y 460.772,Z 323.403,A -85,B 0,C 180,E1 -7917.377,E2 -7917.377} C_VEL
LIN {X 0,Y 460.825,Z 323.391,A -85,B 0,C 180,E1 -7920,E2 -7920} C_VEL
LIN {X 0,Y 460.81,Z 323.398,A -85,B 0,C 180,E1 -7922.622,E2 -7922.622} C_VEL
LIN {X 0,Y 460.695,Z 323.411,A -85,B 0,C 180,E1 -7926.13,E2 -7926.13} C_VEL
LIN {X 0,Y 460.606,Z 323.422,A -85,B 0,C 180,E1 -7928.776,E2 -7928.776} C_VEL
LIN {X 0,Y 460.604,Z 323.423,A -85,B 0,C 180,E1 -7932.334,E2 -7932.334} C_VEL
LIN {X 0,Y 460.597,Z 323.425,A -85,B 0,C 180,E1 -7936.008,E2 -7936.008} C_VEL
LIN {X 0,Y 460.551,Z 323.428,A -85,B 0,C 180,E1 -7938.905,E2 -7938.905} C_VEL
LIN {X 0,Y 460.54,Z 323.433,A -85,B 0,C 180,E1 -7941.484,E2 -7941.484} C_VEL
LIN {X 0,Y 460.527,Z 323.431,A -85,B 0,C 180,E1 -7944.333,E2 -7944.333} C_VEL
LIN {X 0,Y 460.549,Z 323.428,A -85,B 0,C 180,E1 -7947.245,E2 -7947.245} C_VEL
LIN {X 0,Y 460.488,Z 323.439,A -85,B 0,C 180,E1 -7950.241,E2 -7950.241} C_VEL
LIN {X 0,Y 460.508,Z 323.435,A -85,B 0,C 180,E1 -7953.326,E2 -7953.326} C_VEL
LIN {X 0,Y 460.459,Z 323.44,A -85,B 0,C 180,E1 -7956.531,E2 -7956.531} C_VEL
LIN {X 0,Y 460.525,Z 323.433,A -85,B 0,C 180,E1 -7958.9,E2 -7958.9} C_VEL
LIN {X 0,Y 460.503,Z 323.432,A -85,B 0,C 180,E1 -7962.183,E2 -7962.183} C_VEL
LIN {X 0,Y 460.524,Z 323.491,A -85,B 0,C 180,E1 -7965.004,E2 -7965.004} C_VEL
LIN {X 0,Y 464.408,Z 336.047,A -85,B 0,C 180,E1 -7968.255,E2 -7968.255} C_VEL
LIN {X 0,Y 468.162,Z 349.02,A -85,B 0,C 180,E1 -7971.317,E2 -7971.317} C_VEL
LIN {X 0,Y 470.134,Z 357.135,A -85,B 0,C 180,E1 -7973.071,E2 -7973.071} C_VEL
LIN {X 0,Y 469.428,Z 365.329,A -85,B 0,C 180,E1 -7974.543,E2 -7974.543} C_VEL
LIN {X 0,Y 467.711,Z 384.081,A -85,B 0,C 180,E1 -7977.765,E2 -7977.765} C_VEL
LIN {X 0,Y 466.184,Z 403.602,A -85,B 0,C 180,E1 -7980.971,E2 -7980.971} C_VEL
LIN {X 0,Y 465.164,Z 420,A -85,B 0,C 180,E1 -7983.564,E2 -7983.564} C_VEL
LIN {X 0,Y 467.948,Z 432.865,A -85,B 0,C 180,E1 -7983.936,E2 -7983.936} C_VEL
LIN {X 0,Y 470.727,Z 445.838,A -85,B 0,C 180,E1 -7984.347,E2 -7984.347} C_VEL
LIN {X 0,Y 470.05,Z 462.773,A -85,B 0,C 180,E1 -7984.827,E2 -7984.827} C_VEL
LIN {X 0,Y 469.259,Z 478.637,A -85,B 0,C 180,E1 -7985.445,E2 -7985.445} C_VEL
LIN {X 0,Y 468.263,Z 495.085,A -85,B 0,C 180,E1 -7986.28,E2 -7986.28} C_VEL
LIN {X 0,Y 467.205,Z 509.887,A -85,B 0,C 180,E1 -7987.213,E2 -7987.213} C_VEL
LIN {X 0,Y 466.072,Z 524.507,A -85,B 0,C 180,E1 -7988.322,E2 -7988.322} C_VEL
LIN {X 0,Y 465.022,Z 537.136,A -85,B 0,C 180,E1 -7989.475,E2 -7989.475} C_VEL
LIN {X 0,Y 463.913,Z 549.031,A -85,B 0,C 180,E1 -7990.764,E2 -7990.764} C_VEL
LIN {X 0,Y 462.808,Z 561.276,A -85,B 0,C 180,E1 -7992.322,E2 -7992.322} C_VEL
LIN {X 0,Y 462.012,Z 571.975,A -85,B 0,C 180,E1 -7993.928,E2 -7993.928} C_VEL
LIN {X 0,Y 461.148,Z 581.834,A -85,B 0,C 180,E1 -7995.664,E2 -7995.664} C_VEL
LIN {X 0,Y 460.604,Z 589.491,A -85,B 0,C 180,E1 -7997.265,E2 -7997.265} C_VEL
LIN {X 0,Y 460.199,Z 596.5,A -85,B 0,C 180,E1 -7998.997,E2 -7998.997} C_VEL
LIN {X 0,Y 459.859,Z 602.469,A -85,B 0,C 180,E1 -8000.768,E2 -8000.768} C_VEL
LIN {X 0,Y 459.721,Z 608.25,A -85,B 0,C 180,E1 -8002.977,E2 -8002.977} C_VEL
LIN {X 0,Y 459.582,Z 611.637,A -85,B 0,C 180,E1 -8004.738,E2 -8004.738} C_VEL
LIN {X 0,Y 459.533,Z 614.093,A -85,B 0,C 180,E1 -8006.495,E2 -8006.495} C_VEL
LIN {X 0,Y 459.51,Z 615.479,A -85,B 0,C 180,E1 -8008.249,E2 -8008.249} C_VEL
LIN {X 0,Y 459.469,Z 616,A -85,B 0,C 180,E1 -8010.002,E2 -8010.002} C_VEL
LIN {X 0,Y 459.511,Z 615.476,A -85,B 0,C 180,E1 -8011.755,E2 -8011.755} C_VEL
LIN {X 0,Y 459.534,Z 614.087,A -85,B 0,C 180,E1 -8013.509,E2 -8013.509} C_VEL
LIN {X 0,Y 459.584,Z 611.63,A -85,B 0,C 180,E1 -8015.266,E2 -8015.266} C_VEL
LIN {X 0,Y 459.725,Z 608.248,A -85,B 0,C 180,E1 -8017.027,E2 -8017.027} C_VEL
LIN {X 0,Y 459.858,Z 602.461,A -85,B 0,C 180,E1 -8019.236,E2 -8019.236} C_VEL
LIN {X 0,Y 460.27,Z 594.848,A -85,B 0,C 180,E1 -8021.451,E2 -8021.451} C_VEL
LIN {X 0,Y 460.737,Z 587.258,A -85,B 0,C 180,E1 -8023.229,E2 -8023.229} C_VEL
LIN {X 0,Y 461.4,Z 578.196,A -85,B 0,C 180,E1 -8025.009,E2 -8025.009} C_VEL
LIN {X 0,Y 462.255,Z 568.018,A -85,B 0,C 180,E1 -8026.699,E2 -8026.699} C_VEL
LIN {X 0,Y 463.273,Z 556.268,A -85,B 0,C 180,E1 -8028.35,E2 -8028.35} C_VEL
LIN {X 0,Y 464.392,Z 543.38,A -85,B 0,C 180,E1 -8029.879,E2 -8029.879} C_VEL
LIN {X 0,Y 465.626,Z 529.636,A -85,B 0,C 180,E1 -8031.24,E2 -8031.24} C_VEL
LIN {X 0,Y 466.613,Z 517.45,A -85,B 0,C 180,E1 -8032.238,E2 -8032.238} C_VEL
LIN {X 0,Y 467.757,Z 502.939,A -85,B 0,C 180,E1 -8033.234,E2 -8033.234} C_VEL
LIN {X 0,Y 468.735,Z 487.352,A -85,B 0,C 180,E1 -8034.117,E2 -8034.117} C_VEL
LIN {X 0,Y 469.657,Z 471.029,A -85,B 0,C 180,E1 -8034.843,E2 -8034.843} C_VEL
LIN {X 0,Y 470.33,Z 455.286,A -85,B 0,C 180,E1 -8035.377,E2 -8035.377} C_VEL
LIN {X 0,Y 470.551,Z 445.434,A -85,B 0,C 180,E1 -8035.638,E2 -8035.638} C_VEL
LIN {X 0,Y 465.523,Z 422.563,A -85,B 0,C 180,E1 -8036.307,E2 -8036.307} C_VEL
LIN {X 0,Y 465.083,Z 419.731,A -85,B 0,C 180,E1 -8036.386,E2 -8036.386} C_VEL
LIN {X 0,Y 466.107,Z 400.5,A -85,B 0,C 180,E1 -8039.344,E2 -8039.344} C_VEL
LIN {X 0,Y 467.733,Z 379.945,A -85,B 0,C 180,E1 -8042.748,E2 -8042.748} C_VEL
LIN {X 0,Y 469.612,Z 363.832,A -85,B 0,C 180,E1 -8045.71,E2 -8045.71} C_VEL
LIN {X 0,Y 470.408,Z 357.842,A -85,B 0,C 180,E1 -8046.931,E2 -8046.931} C_VEL
LIN {X 0,Y 469.369,Z 352.376,A -85,B 0,C 180,E1 -8048.363,E2 -8048.363} C_VEL
LIN {X 0,Y 467.639,Z 346.344,A -85,B 0,C 180,E1 -8050.26,E2 -8050.26} C_VEL
LIN {X 0,Y 466.003,Z 341.209,A -85,B 0,C 180,E1 -8052.355,E2 -8052.355} C_VEL
LIN {X 0,Y 464.955,Z 338.158,A -85,B 0,C 180,E1 -8054.054,E2 -8054.054} C_VEL
LIN {X 0,Y 464.25,Z 335.969,A -85,B 0,C 180,E1 -8055.864,E2 -8055.864} C_VEL
LIN {X 0,Y 463.783,Z 334.858,A -85,B 0,C 180,E1 -8057.949,E2 -8057.949} C_VEL
LIN {X 0,Y 463.66,Z 334.882,A -85,B 0,C 180,E1 -8059.325,E2 -8059.325} C_VEL
LIN {X 0,Y 463.69,Z 336.03,A -85,B 0,C 180,E1 -8061.58,E2 -8061.58} C_VEL
LIN {X 0,Y 463.86,Z 338.198,A -85,B 0,C 180,E1 -8063.78,E2 -8063.78} C_VEL
LIN {X 0,Y 463.561,Z 341.073,A -85,B 0,C 180,E1 -8065.879,E2 -8065.879} C_VEL
LIN {X 0,Y 462.828,Z 345.896,A -85,B 0,C 180,E1 -8068.917,E2 -8068.917} C_VEL
LIN {X 0,Y 462.426,Z 350.897,A -85,B 0,C 180,E1 -8071.892,E2 -8071.892} C_VEL
LIN {X 0,Y 462.092,Z 355.879,A -85,B 0,C 180,E1 -8074.796,E2 -8074.796} C_VEL
LIN {X 0,Y 461.787,Z 361.786,A -85,B 0,C 180,E1 -8078.184,E2 -8078.184} C_VEL
LIN {X 0,Y 461.479,Z 367.414,A -85,B 0,C 180,E1 -8081.349,E2 -8081.349} C_VEL
LIN {X 0,Y 461.331,Z 371.239,A -85,B 0,C 180,E1 -8083.485,E2 -8083.485} C_VEL
LIN {X 0,Y 465.721,Z 384.52,A -85,B 0,C 180,E1 -8084.239,E2 -8084.239} C_VEL
LIN {X 0,Y 465.334,Z 398.101,A -85,B 0,C 180,E1 -8084.899,E2 -8084.899} C_VEL
LIN {X 0,Y 464.666,Z 409.651,A -85,B 0,C 180,E1 -8085.609,E2 -8085.609} C_VEL
LIN {X 0,Y 464.07,Z 421.623,A -85,B 0,C 180,E1 -8086.536,E2 -8086.536} C_VEL
LIN {X 0,Y 463.407,Z 433.036,A -85,B 0,C 180,E1 -8087.631,E2 -8087.631} C_VEL
LIN {X 0,Y 462.873,Z 443.177,A -85,B 0,C 180,E1 -8088.838,E2 -8088.838} C_VEL
LIN {X 0,Y 462.271,Z 452.19,A -85,B 0,C 180,E1 -8090.152,E2 -8090.152} C_VEL
LIN {X 0,Y 461.773,Z 460.079,A -85,B 0,C 180,E1 -8091.607,E2 -8091.607} C_VEL
LIN {X 0,Y 461.308,Z 466.088,A -85,B 0,C 180,E1 -8093,E2 -8093} C_VEL
LIN {X 0,Y 461.039,Z 470.503,A -85,B 0,C 180,E1 -8094.314,E2 -8094.314} C_VEL
LIN {X 0,Y 460.948,Z 473.815,A -85,B 0,C 180,E1 -8095.628,E2 -8095.628} C_VEL
LIN {X 0,Y 460.803,Z 475.506,A -85,B 0,C 180,E1 -8096.503,E2 -8096.503} C_VEL
LIN {X 0,Y 460.659,Z 476.757,A -85,B 0,C 180,E1 -8097.377,E2 -8097.377} C_VEL
LIN {X 0,Y 460.5,Z 477.59,A -85,B 0,C 180,E1 -8098.251,E2 -8098.251} C_VEL
LIN {X 0,Y 460.449,Z 478.018,A -85,B 0,C 180,E1 -8099.126,E2 -8099.126} C_VEL
LIN {X 0,Y 460.398,Z 478.055,A -85,B 0,C 180,E1 -8100,E2 -8100} C_VEL
LIN {X 0,Y 460.36,Z 477.692,A -85,B 0,C 180,E1 -8100.875,E2 -8100.875} C_VEL
LIN {X 0,Y 460.49,Z 475.694,A -85,B 0,C 180,E1 -8102.625,E2 -8102.625} C_VEL
LIN {X 0,Y 460.522,Z 473.14,A -85,B 0,C 180,E1 -8103.938,E2 -8103.938} C_VEL
LIN {X 0,Y 460.503,Z 469.614,A -85,B 0,C 180,E1 -8105.254,E2 -8105.254} C_VEL
LIN {X 0,Y 460.812,Z 464.226,A -85,B 0,C 180,E1 -8106.756,E2 -8106.756} C_VEL
LIN {X 0,Y 461.013,Z 458.097,A -85,B 0,C 180,E1 -8108.107,E2 -8108.107} C_VEL
LIN {X 0,Y 461.385,Z 450.648,A -85,B 0,C 180,E1 -8109.425,E2 -8109.425} C_VEL
LIN {X 0,Y 461.755,Z 441.436,A -85,B 0,C 180,E1 -8110.746,E2 -8110.746} C_VEL
LIN {X 0,Y 462.289,Z 431.062,A -85,B 0,C 180,E1 -8111.955,E2 -8111.955} C_VEL
LIN {X 0,Y 462.693,Z 420.64,A -85,B 0,C 180,E1 -8112.947,E2 -8112.947} C_VEL
LIN {X 0,Y 463.195,Z 408.266,A -85,B 0,C 180,E1 -8113.895,E2 -8113.895} C_VEL
LIN {X 0,Y 463.743,Z 395.746,A -85,B 0,C 180,E1 -8114.649,E2 -8114.649} C_VEL
LIN {X 0,Y 464.138,Z 382.251,A -85,B 0,C 180,E1 -8115.262,E2 -8115.262} C_VEL
LIN {X 0,Y 461.264,Z 369.523,A -85,B 0,C 180,E1 -8115.802,E2 -8115.802} C_VEL
LIN {X 0,Y 460.178,Z 365.141,A -85,B 0,C 180,E1 -8115.957,E2 -8115.957} C_VEL
LIN {X 0,Y 460.263,Z 359.479,A -85,B 0,C 180,E1 -8118.786,E2 -8118.786} C_VEL
LIN {X 0,Y 460.401,Z 352.265,A -85,B 0,C 180,E1 -8122.435,E2 -8122.435} C_VEL
LIN {X 0,Y 460.546,Z 345.72,A -85,B 0,C 180,E1 -8125.794,E2 -8125.794} C_VEL
LIN {X 0,Y 460.678,Z 341.035,A -85,B 0,C 180,E1 -8128.225,E2 -8128.225} C_VEL
LIN {X 0,Y 460.826,Z 335.087,A -85,B 0,C 180,E1 -8131.343,E2 -8131.343} C_VEL
LIN {X 0,Y 460.983,Z 329.43,A -85,B 0,C 180,E1 -8134.34,E2 -8134.34} C_VEL
LIN {X 0,Y 460.786,Z 325.456,A -85,B 0,C 180,E1 -8136.501,E2 -8136.501} C_VEL
LIN {X 0,Y 460.549,Z 323.434,A -85,B 0,C 180,E1 -8137.619,E2 -8137.619} C_VEL
LIN {X 0,Y 460.536,Z 323.434,A -85,B 0,C 180,E1 -8141.011,E2 -8141.011} C_VEL
LIN {X 0,Y 460.521,Z 323.432,A -85,B 0,C 180,E1 -8144.589,E2 -8144.589} C_VEL
LIN {X 0,Y 460.513,Z 323.437,A -85,B 0,C 180,E1 -8147.816,E2 -8147.816} C_VEL
LIN {X 0,Y 460.527,Z 323.435,A -85,B 0,C 180,E1 -8150.135,E2 -8150.135} C_VEL
LIN {X 0,Y 460.553,Z 323.506,A -85,B 0,C 180,E1 -8152.674,E2 -8152.674} C_VEL
LIN {X 0,Y 461.286,Z 328.216,A -85,B 0,C 180,E1 -8154.621,E2 -8154.621} C_VEL
LIN {X 0,Y 461.3,Z 333.483,A -85,B 0,C 180,E1 -8156.923,E2 -8156.923} C_VEL
LIN {X 0,Y 461.19,Z 339.825,A -85,B 0,C 180,E1 -8159.808,E2 -8159.808} C_VEL
LIN {X 0,Y 461.056,Z 346.995,A -85,B 0,C 180,E1 -8163.275,E2 -8163.275} C_VEL
LIN {X 0,Y 460.968,Z 353.896,A -85,B 0,C 180,E1 -8166.645,E2 -8166.645} C_VEL
LIN {X 0,Y 460.931,Z 359.919,A -85,B 0,C 180,E1 -8169.469,E2 -8169.469} C_VEL
LIN {X 0,Y 460.916,Z 364.764,A -85,B 0,C 180,E1 -8171.614,E2 -8171.614} C_VEL
LIN {X 0,Y 460.274,Z 366.008,A -85,B 0,C 180,E1 -8172.076,E2 -8172.076} C_VEL
LIN {X 0,Y 457.513,Z 368.354,A -85,B 0,C 180,E1 -8172.784,E2 -8172.784} C_VEL
LIN {X 0,Y 454.724,Z 370.765,A -85,B 0,C 180,E1 -8173.498,E2 -8173.498} C_VEL
LIN {X 0,Y 454.064,Z 372.109,A -85,B 0,C 180,E1 -8173.966,E2 -8173.966} C_VEL
LIN {X 0,Y 454.092,Z 372.701,A -85,B 0,C 180,E1 -8174.197,E2 -8174.197} C_VEL
LIN {X 0,Y 457.283,Z 383.511,A -85,B 0,C 180,E1 -8174.596,E2 -8174.596} C_VEL
LIN {X 0,Y 457.069,Z 395.983,A -85,B 0,C 180,E1 -8175.073,E2 -8175.073} C_VEL
LIN {X 0,Y 456.725,Z 408.565,A -85,B 0,C 180,E1 -8175.745,E2 -8175.745} C_VEL
LIN {X 0,Y 456.45,Z 419.454,A -85,B 0,C 180,E1 -8176.515,E2 -8176.515} C_VEL
LIN {X 0,Y 455.987,Z 429.714,A -85,B 0,C 180,E1 -8177.424,E2 -8177.424} C_VEL
LIN {X 0,Y 455.486,Z 438.939,A -85,B 0,C 180,E1 -8178.427,E2 -8178.427} C_VEL
LIN {X 0,Y 455.087,Z 447.343,A -85,B 0,C 180,E1 -8179.543,E2 -8179.543} C_VEL
LIN {X 0,Y 454.587,Z 454.296,A -85,B 0,C 180,E1 -8180.656,E2 -8180.656} C_VEL
LIN {X 0,Y 454.291,Z 461.086,A -85,B 0,C 180,E1 -8181.995,E2 -8181.995} C_VEL
LIN {X 0,Y 453.982,Z 466.487,A -85,B 0,C 180,E1 -8183.331,E2 -8183.331} C_VEL
LIN {X 0,Y 453.579,Z 470.748,A -85,B 0,C 180,E1 -8184.664,E2 -8184.664} C_VEL
LIN {X 0,Y 453.514,Z 472.966,A -85,B 0,C 180,E1 -8185.554,E2 -8185.554} C_VEL
LIN {X 0,Y 453.512,Z 474.768,A -85,B 0,C 180,E1 -8186.444,E2 -8186.444} C_VEL
LIN {X 0,Y 453.396,Z 476.164,A -85,B 0,C 180,E1 -8187.333,E2 -8187.333} C_VEL
LIN {X 0,Y 453.314,Z 477.737,A -85,B 0,C 180,E1 -8189.11,E2 -8189.11} C_VEL
LIN {X 0,Y 453.292,Z 477.971,A -85,B 0,C 180,E1 -8189.998,E2 -8189.998} C_VEL
LIN {X 0,Y 453.328,Z 477.22,A -85,B 0,C 180,E1 -8191.775,E2 -8191.775} C_VEL
LIN {X 0,Y 453.569,Z 474.936,A -85,B 0,C 180,E1 -8193.551,E2 -8193.551} C_VEL
LIN {X 0,Y 453.65,Z 472.153,A -85,B 0,C 180,E1 -8194.886,E2 -8194.886} C_VEL
LIN {X 0,Y 453.842,Z 468.357,A -85,B 0,C 180,E1 -8196.221,E2 -8196.221} C_VEL
LIN {X 0,Y 454.113,Z 463.38,A -85,B 0,C 180,E1 -8197.569,E2 -8197.569} C_VEL
LIN {X 0,Y 454.536,Z 456.032,A -85,B 0,C 180,E1 -8199.117,E2 -8199.117} C_VEL
LIN {X 0,Y 455.026,Z 448.015,A -85,B 0,C 180,E1 -8200.454,E2 -8200.454} C_VEL
LIN {X 0,Y 455.459,Z 439.743,A -85,B 0,C 180,E1 -8201.569,E2 -8201.569} C_VEL
LIN {X 0,Y 455.931,Z 429.565,A -85,B 0,C 180,E1 -8202.686,E2 -8202.686} C_VEL
LIN {X 0,Y 456.455,Z 419.099,A -85,B 0,C 180,E1 -8203.607,E2 -8203.607} C_VEL
LIN {X 0,Y 456.738,Z 408.286,A -85,B 0,C 180,E1 -8204.364,E2 -8204.364} C_VEL
LIN {X 0,Y 457.123,Z 395.611,A -85,B 0,C 180,E1 -8205.034,E2 -8205.034} C_VEL
LIN {X 0,Y 457.145,Z 383.148,A -85,B 0,C 180,E1 -8205.513,E2 -8205.513} C_VEL
LIN {X 0,Y 454.089,Z 372.679,A -85,B 0,C 180,E1 -8205.914,E2 -8205.914} C_VEL
LIN {X 0,Y 453.985,Z 364.599,A -85,B 0,C 180,E1 -8209.208,E2 -8209.208} C_VEL
LIN {X 0,Y 453.996,Z 357.76,A -85,B 0,C 180,E1 -8212.285,E2 -8212.285} C_VEL
LIN {X 0,Y 454.006,Z 352.714,A -85,B 0,C 180,E1 -8214.703,E2 -8214.703} C_VEL
LIN {X 0,Y 454.107,Z 346.651,A -85,B 0,C 180,E1 -8217.662,E2 -8217.662} C_VEL
LIN {X 0,Y 454.27,Z 340.311,A -85,B 0,C 180,E1 -8220.697,E2 -8220.697} C_VEL
LIN {X 0,Y 454.415,Z 333.427,A -85,B 0,C 180,E1 -8223.83,E2 -8223.83} C_VEL
LIN {X 0,Y 454.189,Z 328.353,A -85,B 0,C 180,E1 -8226.012,E2 -8226.012} C_VEL
LIN {X 0,Y 453.456,Z 324.316,A -85,B 0,C 180,E1 -8227.773,E2 -8227.773} C_VEL
LIN {X 0,Y 453.48,Z 324.311,A -85,B 0,C 180,E1 -8230.607,E2 -8230.607} C_VEL
LIN {X 0,Y 453.448,Z 324.313,A -85,B 0,C 180,E1 -8234.219,E2 -8234.219} C_VEL
LIN {X 0,Y 453.477,Z 324.314,A -85,B 0,C 180,E1 -8237.006,E2 -8237.006} C_VEL
LIN {X 0,Y 453.521,Z 324.308,A -85,B 0,C 180,E1 -8240.553,E2 -8240.553} C_VEL
LIN {X 0,Y 453.439,Z 324.316,A -85,B 0,C 180,E1 -8243.915,E2 -8243.915} C_VEL
LIN {X 0,Y 453.463,Z 324.311,A -85,B 0,C 180,E1 -8247.149,E2 -8247.149} C_VEL
LIN {X 0,Y 453.454,Z 324.309,A -85,B 0,C 180,E1 -8250.266,E2 -8250.266} C_VEL
LIN {X 0,Y 453.494,Z 324.302,A -85,B 0,C 180,E1 -8253.293,E2 -8253.293} C_VEL
LIN {X 0,Y 453.497,Z 324.307,A -85,B 0,C 180,E1 -8256.238,E2 -8256.238} C_VEL
LIN {X 0,Y 453.496,Z 324.307,A -85,B 0,C 180,E1 -8259.118,E2 -8259.118} C_VEL
LIN {X 0,Y 453.488,Z 324.306,A -85,B 0,C 180,E1 -8261.943,E2 -8261.943} C_VEL
LIN {X 0,Y 453.516,Z 324.306,A -85,B 0,C 180,E1 -8264.725,E2 -8264.725} C_VEL
LIN {X 0,Y 453.573,Z 324.301,A -85,B 0,C 180,E1 -8268.379,E2 -8268.379} C_VEL
LIN {X 0,Y 453.628,Z 324.293,A -85,B 0,C 180,E1 -8271.984,E2 -8271.984} C_VEL
LIN {X 0,Y 453.649,Z 324.285,A -85,B 0,C 180,E1 -8274.666,E2 -8274.666} C_VEL
LIN {X 0,Y 453.716,Z 324.282,A -85,B 0,C 180,E1 -8277.336,E2 -8277.336} C_VEL
LIN {X 0,Y 453.796,Z 324.266,A -85,B 0,C 180,E1 -8280,E2 -8280} C_VEL
LIN {X 0,Y 453.751,Z 324.277,A -85,B 0,C 180,E1 -8282.663,E2 -8282.663} C_VEL
LIN {X 0,Y 453.661,Z 324.287,A -85,B 0,C 180,E1 -8286.225,E2 -8286.225} C_VEL
LIN {X 0,Y 453.57,Z 324.299,A -85,B 0,C 180,E1 -8288.913,E2 -8288.913} C_VEL
LIN {X 0,Y 453.576,Z 324.3,A -85,B 0,C 180,E1 -8292.551,E2 -8292.551} C_VEL
LIN {X 0,Y 453.533,Z 324.307,A -85,B 0,C 180,E1 -8296.196,E2 -8296.196} C_VEL
LIN {X 0,Y 453.5,Z 324.306,A -85,B 0,C 180,E1 -8299.043,E2 -8299.043} C_VEL
LIN {X 0,Y 453.481,Z 324.311,A -85,B 0,C 180,E1 -8301.836,E2 -8301.836} C_VEL
LIN {X 0,Y 453.495,Z 324.309,A -85,B 0,C 180,E1 -8304.735,E2 -8304.735} C_VEL
LIN {X 0,Y 453.508,Z 324.305,A -85,B 0,C 180,E1 -8307.961,E2 -8307.961} C_VEL
LIN {X 0,Y 453.444,Z 324.315,A -85,B 0,C 180,E1 -8311.527,E2 -8311.527} C_VEL
LIN {X 0,Y 453.468,Z 324.312,A -85,B 0,C 180,E1 -8314.779,E2 -8314.779} C_VEL
LIN {X 0,Y 453.453,Z 324.313,A -85,B 0,C 180,E1 -8318.312,E2 -8318.312} C_VEL
LIN {X 0,Y 453.474,Z 324.312,A -85,B 0,C 180,E1 -8320.611,E2 -8320.611} C_VEL
LIN {X 0,Y 453.436,Z 324.312,A -85,B 0,C 180,E1 -8323.246,E2 -8323.246} C_VEL
LIN {X 0,Y 453.48,Z 324.44,A -85,B 0,C 180,E1 -8324.336,E2 -8324.336} C_VEL
LIN {X 0,Y 457.206,Z 336.503,A -85,B 0,C 180,E1 -8327.547,E2 -8327.547} C_VEL
LIN {X 0,Y 460.268,Z 346.952,A -85,B 0,C 180,E1 -8330.114,E2 -8330.114} C_VEL
LIN {X 0,Y 463.033,Z 357.056,A -85,B 0,C 180,E1 -8332.413,E2 -8332.413} C_VEL
LIN {X 0,Y 463.52,Z 360.783,A -85,B 0,C 180,E1 -8333.185,E2 -8333.185} C_VEL
LIN {X 0,Y 461.667,Z 377.953,A -85,B 0,C 180,E1 -8336.248,E2 -8336.248} C_VEL
LIN {X 0,Y 460.01,Z 396.839,A -85,B 0,C 180,E1 -8339.473,E2 -8339.473} C_VEL
LIN {X 0,Y 458.488,Z 416.901,A -85,B 0,C 180,E1 -8342.755,E2 -8342.755} C_VEL
LIN {X 0,Y 458.304,Z 419.666,A -85,B 0,C 180,E1 -8343.19,E2 -8343.19} C_VEL
LIN {X 0,Y 461.576,Z 434.993,A -85,B 0,C 180,E1 -8343.653,E2 -8343.653} C_VEL
LIN {X 0,Y 464.115,Z 447.078,A -85,B 0,C 180,E1 -8344.055,E2 -8344.055} C_VEL
LIN {X 0,Y 463.335,Z 464.393,A -85,B 0,C 180,E1 -8344.577,E2 -8344.577} C_VEL
LIN {X 0,Y 462.367,Z 481.586,A -85,B 0,C 180,E1 -8345.294,E2 -8345.294} C_VEL
LIN {X 0,Y 461.412,Z 496.525,A -85,B 0,C 180,E1 -8346.091,E2 -8346.091} C_VEL
LIN {X 0,Y 460.26,Z 511.714,A -85,B 0,C 180,E1 -8347.087,E2 -8347.087} C_VEL
LIN {X 0,Y 459.094,Z 525.886,A -85,B 0,C 180,E1 -8348.211,E2 -8348.211} C_VEL
LIN {X 0,Y 457.932,Z 538.822,A -85,B 0,C 180,E1 -8349.419,E2 -8349.419} C_VEL
LIN {X 0,Y 456.933,Z 550.579,A -85,B 0,C 180,E1 -8350.692,E2 -8350.692} C_VEL
LIN {X 0,Y 455.95,Z 561.233,A -85,B 0,C 180,E1 -8352.047,E2 -8352.047} C_VEL
LIN {X 0,Y 455.059,Z 572.002,A -85,B 0,C 180,E1 -8353.681,E2 -8353.681} C_VEL
LIN {X 0,Y 454.174,Z 581.834,A -85,B 0,C 180,E1 -8355.439,E2 -8355.439} C_VEL
LIN {X 0,Y 453.619,Z 589.289,A -85,B 0,C 180,E1 -8357.02,E2 -8357.02} C_VEL
LIN {X 0,Y 453.167,Z 596.499,A -85,B 0,C 180,E1 -8358.824,E2 -8358.824} C_VEL
LIN {X 0,Y 452.791,Z 602.469,A -85,B 0,C 180,E1 -8360.623,E2 -8360.623} C_VEL
LIN {X 0,Y 452.643,Z 608.25,A -85,B 0,C 180,E1 -8362.867,E2 -8362.867} C_VEL
LIN {X 0,Y 452.499,Z 611.637,A -85,B 0,C 180,E1 -8364.655,E2 -8364.655} C_VEL
LIN {X 0,Y 452.43,Z 614.093,A -85,B 0,C 180,E1 -8366.44,E2 -8366.44} C_VEL
LIN {X 0,Y 452.426,Z 615.479,A -85,B 0,C 180,E1 -8368.222,E2 -8368.222} C_VEL
LIN {X 0,Y 452.377,Z 616,A -85,B 0,C 180,E1 -8370.002,E2 -8370.002} C_VEL
LIN {X 0,Y 452.427,Z 615.476,A -85,B 0,C 180,E1 -8371.782,E2 -8371.782} C_VEL
LIN {X 0,Y 452.431,Z 614.087,A -85,B 0,C 180,E1 -8373.564,E2 -8373.564} C_VEL
LIN {X 0,Y 452.501,Z 611.629,A -85,B 0,C 180,E1 -8375.349,E2 -8375.349} C_VEL
LIN {X 0,Y 452.647,Z 608.248,A -85,B 0,C 180,E1 -8377.137,E2 -8377.137} C_VEL
LIN {X 0,Y 452.791,Z 602.461,A -85,B 0,C 180,E1 -8379.382,E2 -8379.382} C_VEL
LIN {X 0,Y 453.242,Z 594.848,A -85,B 0,C 180,E1 -8381.631,E2 -8381.631} C_VEL
LIN {X 0,Y 453.825,Z 586.249,A -85,B 0,C 180,E1 -8383.662,E2 -8383.662} C_VEL
LIN {X 0,Y 454.62,Z 576.964,A -85,B 0,C 180,E1 -8385.468,E2 -8385.468} C_VEL
LIN {X 0,Y 455.434,Z 567.408,A -85,B 0,C 180,E1 -8387.051,E2 -8387.051} C_VEL
LIN {X 0,Y 456.275,Z 557.873,A -85,B 0,C 180,E1 -8388.409,E2 -8388.409} C_VEL
LIN {X 0,Y 457.247,Z 546.425,A -85,B 0,C 180,E1 -8389.766,E2 -8389.766} C_VEL
LIN {X 0,Y 458.442,Z 533.068,A -85,B 0,C 180,E1 -8391.118,E2 -8391.118} C_VEL
LIN {X 0,Y 459.636,Z 518.58,A -85,B 0,C 180,E1 -8392.357,E2 -8392.357} C_VEL
LIN {X 0,Y 460.875,Z 503.45,A -85,B 0,C 180,E1 -8393.433,E2 -8393.433} C_VEL
LIN {X 0,Y 461.867,Z 488.239,A -85,B 0,C 180,E1 -8394.319,E2 -8394.319} C_VEL
LIN {X 0,Y 462.798,Z 472.697,A -85,B 0,C 180,E1 -8395.045,E2 -8395.045} C_VEL
LIN {X 0,Y 463.581,Z 457.092,A -85,B 0,C 180,E1 -8395.611,E2 -8395.611} C_VEL
LIN {X 0,Y 463.864,Z 446.546,A -85,B 0,C 180,E1 -8395.908,E2 -8395.908} C_VEL
LIN {X 0,Y 459.801,Z 428.186,A -85,B 0,C 180,E1 -8396.49,E2 -8396.49} C_VEL
LIN {X 0,Y 458.201,Z 419.151,A -85,B 0,C 180,E1 -8396.737,E2 -8396.737} C_VEL
LIN {X 0,Y 459.394,Z 399.841,A -85,B 0,C 180,E1 -8399.817,E2 -8399.817} C_VEL
LIN {X 0,Y 460.81,Z 382.844,A -85,B 0,C 180,E1 -8402.688,E2 -8402.688} C_VEL
LIN {X 0,Y 462.694,Z 367.697,A -85,B 0,C 180,E1 -8405.522,E2 -8405.522} C_VEL
LIN {X 0,Y 463.823,Z 360.266,A -85,B 0,C 180,E1 -8407.057,E2 -8407.057} C_VEL
LIN {X 0,Y 462.605,Z 354.105,A -85,B 0,C 180,E1 -8408.741,E2 -8408.741} C_VEL
LIN {X 0,Y 461.171,Z 349.203,A -85,B 0,C 180,E1 -8410.362,E2 -8410.362} C_VEL
LIN {X 0,Y 459.726,Z 344.566,A -85,B 0,C 180,E1 -8412.273,E2 -8412.273} C_VEL
LIN {X 0,Y 458.691,Z 341.548,A -85,B 0,C 180,E1 -8413.935,E2 -8413.935} C_VEL
LIN {X 0,Y 458.156,Z 339.939,A -85,B 0,C 180,E1 -8415.12,E2 -8415.12} C_VEL
LIN {X 0,Y 457.751,Z 338.792,A -85,B 0,C 180,E1 -8416.299,E2 -8416.299} C_VEL
LIN {X 0,Y 457.443,Z 338.081,A -85,B 0,C 180,E1 -8417.517,E2 -8417.517} C_VEL
LIN {X 0,Y 457.181,Z 337.935,A -85,B 0,C 180,E1 -8419.786,E2 -8419.786} C_VEL
LIN {X 0,Y 457.17,Z 339.136,A -85,B 0,C 180,E1 -8422.055,E2 -8422.055} C_VEL
LIN {X 0,Y 457.228,Z 340.103,A -85,B 0,C 180,E1 -8423.169,E2 -8423.169} C_VEL
LIN {X 0,Y 456.952,Z 342.667,A -85,B 0,C 180,E1 -8425.315,E2 -8425.315} C_VEL
LIN {X 0,Y 456.141,Z 347.248,A -85,B 0,C 180,E1 -8428.409,E2 -8428.409} C_VEL
LIN {X 0,Y 455.612,Z 352.307,A -85,B 0,C 180,E1 -8431.554,E2 -8431.554} C_VEL
LIN {X 0,Y 455.257,Z 357.038,A -85,B 0,C 180,E1 -8434.39,E2 -8434.39} C_VEL
LIN {X 0,Y 454.914,Z 363.119,A -85,B 0,C 180,E1 -8437.966,E2 -8437.966} C_VEL
LIN {X 0,Y 454.588,Z 368.54,A -85,B 0,C 180,E1 -8441.055,E2 -8441.055} C_VEL
LIN {X 0,Y 454.453,Z 372.345,A -85,B 0,C 180,E1 -8443.118,E2 -8443.118} C_VEL
LIN {X 0,Y 458.921,Z 385.272,A -85,B 0,C 180,E1 -8443.885,E2 -8443.885} C_VEL
LIN {X 0,Y 459.265,Z 387.631,A -85,B 0,C 180,E1 -8444.012,E2 -8444.012} C_VEL
LIN {X 0,Y 458.669,Z 400.501,A -85,B 0,C 180,E1 -8444.674,E2 -8444.674} C_VEL
LIN {X 0,Y 457.947,Z 413.53,A -85,B 0,C 180,E1 -8445.528,E2 -8445.528} C_VEL
LIN {X 0,Y 457.297,Z 424.725,A -85,B 0,C 180,E1 -8446.446,E2 -8446.446} C_VEL
LIN {X 0,Y 456.586,Z 435.707,A -85,B 0,C 180,E1 -8447.556,E2 -8447.556} C_VEL
LIN {X 0,Y 456.066,Z 444.723,A -85,B 0,C 180,E1 -8448.669,E2 -8448.669} C_VEL
LIN {X 0,Y 455.44,Z 453.646,A -85,B 0,C 180,E1 -8450.003,E2 -8450.003} C_VEL
LIN {X 0,Y 454.95,Z 460.978,A -85,B 0,C 180,E1 -8451.37,E2 -8451.37} C_VEL
LIN {X 0,Y 454.398,Z 467.474,A -85,B 0,C 180,E1 -8452.893,E2 -8452.893} C_VEL
LIN {X 0,Y 454.128,Z 471.839,A -85,B 0,C 180,E1 -8454.227,E2 -8454.227} C_VEL
LIN {X 0,Y 453.988,Z 475.114,A -85,B 0,C 180,E1 -8455.561,E2 -8455.561} C_VEL
LIN {X 0,Y 453.833,Z 476.783,A -85,B 0,C 180,E1 -8456.449,E2 -8456.449} C_VEL
LIN {X 0,Y 453.696,Z 478.013,A -85,B 0,C 180,E1 -8457.337,E2 -8457.337} C_VEL
LIN {X 0,Y 453.527,Z 478.827,A -85,B 0,C 180,E1 -8458.224,E2 -8458.224} C_VEL
LIN {X 0,Y 453.463,Z 479.232,A -85,B 0,C 180,E1 -8459.112,E2 -8459.112} C_VEL
LIN {X 0,Y 453.411,Z 479.25,A -85,B 0,C 180,E1 -8460,E2 -8460} C_VEL
LIN {X 0,Y 453.382,Z 478.861,A -85,B 0,C 180,E1 -8460.889,E2 -8460.889} C_VEL
LIN {X 0,Y 453.422,Z 478.037,A -85,B 0,C 180,E1 -8461.777,E2 -8461.777} C_VEL
LIN {X 0,Y 453.502,Z 476.815,A -85,B 0,C 180,E1 -8462.665,E2 -8462.665} C_VEL
LIN {X 0,Y 453.519,Z 474.219,A -85,B 0,C 180,E1 -8463.999,E2 -8463.999} C_VEL
LIN {X 0,Y 453.508,Z 470.641,A -85,B 0,C 180,E1 -8465.336,E2 -8465.336} C_VEL
LIN {X 0,Y 453.834,Z 465.593,A -85,B 0,C 180,E1 -8466.759,E2 -8466.759} C_VEL
LIN {X 0,Y 454.056,Z 458.999,A -85,B 0,C 180,E1 -8468.232,E2 -8468.232} C_VEL
LIN {X 0,Y 454.451,Z 451.486,A -85,B 0,C 180,E1 -8469.57,E2 -8469.57} C_VEL
LIN {X 0,Y 454.821,Z 442.221,A -85,B 0,C 180,E1 -8470.912,E2 -8470.912} C_VEL
LIN {X 0,Y 455.405,Z 431.786,A -85,B 0,C 180,E1 -8472.138,E2 -8472.138} C_VEL
LIN {X 0,Y 455.831,Z 421.318,A -85,B 0,C 180,E1 -8473.145,E2 -8473.145} C_VEL
LIN {X 0,Y 456.35,Z 408.801,A -85,B 0,C 180,E1 -8474.116,E2 -8474.116} C_VEL
LIN {X 0,Y 456.932,Z 396.405,A -85,B 0,C 180,E1 -8474.873,E2 -8474.873} C_VEL
LIN {X 0,Y 457.226,Z 382.559,A -85,B 0,C 180,E1 -8475.516,E2 -8475.516} C_VEL
LIN {X 0,Y 454.041,Z 369.246,A -85,B 0,C 180,E1 -8476.092,E2 -8476.092} C_VEL
LIN {X 0,Y 453.135,Z 365.483,A -85,B 0,C 180,E1 -8476.24,E2 -8476.24} C_VEL
LIN {X 0,Y 453.222,Z 360.003,A -85,B 0,C 180,E1 -8479.005,E2 -8479.005} C_VEL
LIN {X 0,Y 453.351,Z 354.41,A -85,B 0,C 180,E1 -8481.843,E2 -8481.843} C_VEL
LIN {X 0,Y 453.464,Z 348.783,A -85,B 0,C 180,E1 -8484.738,E2 -8484.738} C_VEL
LIN {X 0,Y 453.64,Z 342.568,A -85,B 0,C 180,E1 -8487.983,E2 -8487.983} C_VEL
LIN {X 0,Y 453.792,Z 337.333,A -85,B 0,C 180,E1 -8490.736,E2 -8490.736} C_VEL
LIN {X 0,Y 453.934,Z 331.455,A -85,B 0,C 180,E1 -8493.874,E2 -8493.874} C_VEL
LIN {X 0,Y 453.817,Z 326.904,A -85,B 0,C 180,E1 -8496.36,E2 -8496.36} C_VEL
LIN {X 0,Y 453.496,Z 324.313,A -85,B 0,C 180,E1 -8497.855,E2 -8497.855} C_VEL
LIN {X 0,Y 453.502,Z 324.31,A -85,B 0,C 180,E1 -8500.609,E2 -8500.609} C_VEL
LIN {X 0,Y 453.469,Z 324.312,A -85,B 0,C 180,E1 -8504.221,E2 -8504.221} C_VEL
LIN {X 0,Y 453.457,Z 324.315,A -85,B 0,C 180,E1 -8507.003,E2 -8507.003} C_VEL
LIN {X 0,Y 453.502,Z 324.309,A -85,B 0,C 180,E1 -8509.408,E2 -8509.408} C_VEL
LIN {X 0,Y 453.522,Z 324.338,A -85,B 0,C 180,E1 -8512.443,E2 -8512.443} C_VEL
LIN {X 0,Y 454.306,Z 329.409,A -85,B 0,C 180,E1 -8514.54,E2 -8514.54} C_VEL
LIN {X 0,Y 454.335,Z 334.186,A -85,B 0,C 180,E1 -8516.649,E2 -8516.649} C_VEL
LIN {X 0,Y 454.259,Z 340.064,A -85,B 0,C 180,E1 -8519.297,E2 -8519.297} C_VEL
LIN {X 0,Y 454.087,Z 347.429,A -85,B 0,C 180,E1 -8522.832,E2 -8522.832} C_VEL
LIN {X 0,Y 453.99,Z 354.495,A -85,B 0,C 180,E1 -8526.264,E2 -8526.264} C_VEL
LIN {X 0,Y 453.986,Z 360.646,A -85,B 0,C 180,E1 -8529.14,E2 -8529.14} C_VEL
LIN {X 0,Y 454.005,Z 368.244,A -85,B 0,C 180,E1 -8532.429,E2 -8532.429} C_VEL
LIN {X 0,Y 454.064,Z 372.109,A -85,B 0,C 180,E1 -8533.966,E2 -8533.966} C_VEL
LIN {X 0,Y 454.773,Z 373.107,A -85,B 0,C 180,E1 -8534.18,E2 -8534.18} C_VEL
LIN {X 0,Y 456.856,Z 375.318,A -85,B 0,C 180,E1 -8534.364,E2 -8534.364} C_VEL
LIN {X 0,Y 458.037,Z 377.755,A -85,B 0,C 180,E1 -8534.463,E2 -8534.463} C_VEL
LIN {X 0,Y 457.695,Z 380.071,A -85,B 0,C 180,E1 -8534.507,E2 -8534.507} C_VEL
LIN {X 0,Y 454.255,Z 385.987,A -85,B 0,C 180,E1 -8534.56,E2 -8534.56} C_VEL
LIN {X 0,Y 453.404,Z 391.963,A -85,B 0,C 180,E1 -8534.741,E2 -8534.741} C_VEL
LIN {X 0,Y 450.731,Z 399.582,A -85,B 0,C 180,E1 -8534.964,E2 -8534.964} C_VEL
LIN {X 0,Y 450.162,Z 402.389,A -85,B 0,C 180,E1 -8535.109,E2 -8535.109} C_VEL
LIN {X 0,Y 449.797,Z 413.938,A -85,B 0,C 180,E1 -8535.812,E2 -8535.812} C_VEL
LIN {X 0,Y 449.372,Z 424.788,A -85,B 0,C 180,E1 -8536.661,E2 -8536.661} C_VEL
LIN {X 0,Y 448.897,Z 435.116,A -85,B 0,C 180,E1 -8537.681,E2 -8537.681} C_VEL
LIN {X 0,Y 448.348,Z 445.274,A -85,B 0,C 180,E1 -8538.927,E2 -8538.927} C_VEL
LIN {X 0,Y 447.796,Z 454.069,A -85,B 0,C 180,E1 -8540.285,E2 -8540.285} C_VEL
LIN {X 0,Y 447.41,Z 460.055,A -85,B 0,C 180,E1 -8541.416,E2 -8541.416} C_VEL
LIN {X 0,Y 447.154,Z 465.877,A -85,B 0,C 180,E1 -8542.775,E2 -8542.775} C_VEL
LIN {X 0,Y 446.664,Z 470.524,A -85,B 0,C 180,E1 -8544.128,E2 -8544.128} C_VEL
LIN {X 0,Y 446.518,Z 474.043,A -85,B 0,C 180,E1 -8545.484,E2 -8545.484} C_VEL
LIN {X 0,Y 446.52,Z 475.843,A -85,B 0,C 180,E1 -8546.388,E2 -8546.388} C_VEL
LIN {X 0,Y 446.389,Z 477.24,A -85,B 0,C 180,E1 -8547.291,E2 -8547.291} C_VEL
LIN {X 0,Y 446.302,Z 478.813,A -85,B 0,C 180,E1 -8549.096,E2 -8549.096} C_VEL
LIN {X 0,Y 446.277,Z 479.048,A -85,B 0,C 180,E1 -8549.998,E2 -8549.998} C_VEL
LIN {X 0,Y 446.329,Z 478.294,A -85,B 0,C 180,E1 -8551.802,E2 -8551.802} C_VEL
LIN {X 0,Y 446.569,Z 476.011,A -85,B 0,C 180,E1 -8553.607,E2 -8553.607} C_VEL
LIN {X 0,Y 446.657,Z 473.228,A -85,B 0,C 180,E1 -8554.962,E2 -8554.962} C_VEL
LIN {X 0,Y 446.87,Z 469.43,A -85,B 0,C 180,E1 -8556.318,E2 -8556.318} C_VEL
LIN {X 0,Y 447.184,Z 464.298,A -85,B 0,C 180,E1 -8557.723,E2 -8557.723} C_VEL
LIN {X 0,Y 447.607,Z 457.102,A -85,B 0,C 180,E1 -8559.259,E2 -8559.259} C_VEL
LIN {X 0,Y 448.135,Z 449.081,A -85,B 0,C 180,E1 -8560.616,E2 -8560.616} C_VEL
LIN {X 0,Y 448.592,Z 440.807,A -85,B 0,C 180,E1 -8561.749,E2 -8561.749} C_VEL
LIN {X 0,Y 449.087,Z 430.626,A -85,B 0,C 180,E1 -8562.883,E2 -8562.883} C_VEL
LIN {X 0,Y 449.633,Z 420.136,A -85,B 0,C 180,E1 -8563.819,E2 -8563.819} C_VEL
LIN {X 0,Y 449.934,Z 409.333,A -85,B 0,C 180,E1 -8564.586,E2 -8564.586} C_VEL
LIN {X 0,Y 450.339,Z 396.644,A -85,B 0,C 180,E1 -8565.266,E2 -8565.266} C_VEL
LIN {X 0,Y 450.392,Z 384.597,A -85,B 0,C 180,E1 -8565.738,E2 -8565.738} C_VEL
LIN {X 0,Y 447.169,Z 373.683,A -85,B 0,C 180,E1 -8566.157,E2 -8566.157} C_VEL
LIN {X 0,Y 447.046,Z 365.698,A -85,B 0,C 180,E1 -8569.393,E2 -8569.393} C_VEL
LIN {X 0,Y 447.033,Z 358.431,A -85,B 0,C 180,E1 -8572.652,E2 -8572.652} C_VEL
LIN {X 0,Y 447.092,Z 352.283,A -85,B 0,C 180,E1 -8575.609,E2 -8575.609} C_VEL
LIN {X 0,Y 447.148,Z 346.616,A -85,B 0,C 180,E1 -8578.336,E2 -8578.336} C_VEL
LIN {X 0,Y 447.324,Z 340.537,A -85,B 0,C 180,E1 -8581.226,E2 -8581.226} C_VEL
LIN {X 0,Y 447.447,Z 333.442,A -85,B 0,C 180,E1 -8584.43,E2 -8584.43} C_VEL
LIN {X 0,Y 447.223,Z 329.543,A -85,B 0,C 180,E1 -8586.104,E2 -8586.104} C_VEL
LIN {X 0,Y 446.417,Z 325.194,A -85,B 0,C 180,E1 -8588.002,E2 -8588.002} C_VEL
LIN {X 0,Y 446.409,Z 325.192,A -85,B 0,C 180,E1 -8590.914,E2 -8590.914} C_VEL
LIN {X 0,Y 446.386,Z 325.195,A -85,B 0,C 180,E1 -8593.844,E2 -8593.844} C_VEL
LIN {X 0,Y 446.432,Z 325.187,A -85,B 0,C 180,E1 -8596.394,E2 -8596.394} C_VEL
LIN {X 0,Y 446.454,Z 325.184,A -85,B 0,C 180,E1 -8599.803,E2 -8599.803} C_VEL
LIN {X 0,Y 446.418,Z 325.19,A -85,B 0,C 180,E1 -8602.122,E2 -8602.122} C_VEL
LIN {X 0,Y 446.412,Z 325.192,A -85,B 0,C 180,E1 -8605.475,E2 -8605.475} C_VEL
LIN {X 0,Y 446.395,Z 325.193,A -85,B 0,C 180,E1 -8608.698,E2 -8608.698} C_VEL
LIN {X 0,Y 446.464,Z 325.183,A -85,B 0,C 180,E1 -8611.82,E2 -8611.82} C_VEL
LIN {X 0,Y 446.454,Z 325.185,A -85,B 0,C 180,E1 -8614.847,E2 -8614.847} C_VEL
LIN {X 0,Y 446.463,Z 325.185,A -85,B 0,C 180,E1 -8618.231,E2 -8618.231} C_VEL
LIN {X 0,Y 446.434,Z 325.185,A -85,B 0,C 180,E1 -8621.648,E2 -8621.648} C_VEL
LIN {X 0,Y 446.484,Z 325.181,A -85,B 0,C 180,E1 -8624.479,E2 -8624.479} C_VEL
LIN {X 0,Y 446.529,Z 325.178,A -85,B 0,C 180,E1 -8628.193,E2 -8628.193} C_VEL
LIN {X 0,Y 446.577,Z 325.169,A -85,B 0,C 180,E1 -8631.857,E2 -8631.857} C_VEL
LIN {X 0,Y 446.624,Z 325.16,A -85,B 0,C 180,E1 -8634.582,E2 -8634.582} C_VEL
LIN {X 0,Y 446.638,Z 325.161,A -85,B 0,C 180,E1 -8638.196,E2 -8638.196} C_VEL
LIN {X 0,Y 446.766,Z 325.142,A -85,B 0,C 180,E1 -8640,E2 -8640} C_VEL
LIN {X 0,Y 446.695,Z 325.156,A -85,B 0,C 180,E1 -8642.705,E2 -8642.705} C_VEL
LIN {X 0,Y 446.629,Z 325.162,A -85,B 0,C 180,E1 -8646.324,E2 -8646.324} C_VEL
LIN {X 0,Y 446.516,Z 325.179,A -85,B 0,C 180,E1 -8649.055,E2 -8649.055} C_VEL
LIN {X 0,Y 446.508,Z 325.181,A -85,B 0,C 180,E1 -8652.73,E2 -8652.73} C_VEL
LIN {X 0,Y 446.473,Z 325.185,A -85,B 0,C 180,E1 -8656.459,E2 -8656.459} C_VEL
LIN {X 0,Y 446.448,Z 325.186,A -85,B 0,C 180,E1 -8659.304,E2 -8659.304} C_VEL
LIN {X 0,Y 446.42,Z 325.189,A -85,B 0,C 180,E1 -8662.199,E2 -8662.199} C_VEL
LIN {X 0,Y 446.437,Z 325.189,A -85,B 0,C 180,E1 -8665.153,E2 -8665.153} C_VEL
LIN {X 0,Y 446.461,Z 325.184,A -85,B 0,C 180,E1 -8668.18,E2 -8668.18} C_VEL
LIN {X 0,Y 446.398,Z 325.194,A -85,B 0,C 180,E1 -8671.777,E2 -8671.777} C_VEL
LIN {X 0,Y 446.409,Z 325.191,A -85,B 0,C 180,E1 -8674.524,E2 -8674.524} C_VEL
LIN {X 0,Y 446.411,Z 325.19,A -85,B 0,C 180,E1 -8678.084,E2 -8678.084} C_VEL
LIN {X 0,Y 446.407,Z 325.189,A -85,B 0,C 180,E1 -8680.919,E2 -8680.919} C_VEL
LIN {X 0,Y 446.418,Z 325.32,A -85,B 0,C 180,E1 -8683.642,E2 -8683.642} C_VEL
LIN {X 0,Y 449.932,Z 336.528,A -85,B 0,C 180,E1 -8686.717,E2 -8686.717} C_VEL
LIN {X 0,Y 453.459,Z 348.591,A -85,B 0,C 180,E1 -8689.756,E2 -8689.756} C_VEL
LIN {X 0,Y 456.055,Z 357.947,A -85,B 0,C 180,E1 -8691.949,E2 -8691.949} C_VEL
LIN {X 0,Y 456.907,Z 362.169,A -85,B 0,C 180,E1 -8692.867,E2 -8692.867} C_VEL
LIN {X 0,Y 455.343,Z 376.251,A -85,B 0,C 180,E1 -8695.447,E2 -8695.447} C_VEL
LIN {X 0,Y 453.555,Z 394.103,A -85,B 0,C 180,E1 -8698.586,E2 -8698.586} C_VEL
LIN {X 0,Y 451.921,Z 413.997,A -85,B 0,C 180,E1 -8701.941,E2 -8701.941} C_VEL
LIN {X 0,Y 451.505,Z 419.326,A -85,B 0,C 180,E1 -8702.817,E2 -8702.817} C_VEL
LIN {X 0,Y 454.945,Z 435.96,A -85,B 0,C 180,E1 -8703.325,E2 -8703.325} C_VEL
LIN {X 0,Y 457.479,Z 448.335,A -85,B 0,C 180,E1 -8703.755,E2 -8703.755} C_VEL
LIN {X 0,Y 456.681,Z 465.143,A -85,B 0,C 180,E1 -8704.288,E2 -8704.288} C_VEL
LIN {X 0,Y 455.64,Z 482.21,A -85,B 0,C 180,E1 -8705.027,E2 -8705.027} C_VEL
LIN {X 0,Y 454.544,Z 498.222,A -85,B 0,C 180,E1 -8705.92,E2 -8705.92} C_VEL
LIN {X 0,Y 453.276,Z 513.356,A -85,B 0,C 180,E1 -8706.955,E2 -8706.955} C_VEL
LIN {X 0,Y 452.09,Z 527.228,A -85,B 0,C 180,E1 -8708.096,E2 -8708.096} C_VEL
LIN {X 0,Y 450.751,Z 541.344,A -85,B 0,C 180,E1 -8709.48,E2 -8709.48} C_VEL
LIN {X 0,Y 449.684,Z 553.131,A -85,B 0,C 180,E1 -8710.843,E2 -8710.843} C_VEL
LIN {X 0,Y 448.611,Z 565.076,A -85,B 0,C 180,E1 -8712.451,E2 -8712.451} C_VEL
LIN {X 0,Y 447.818,Z 575.324,A -85,B 0,C 180,E1 -8714.062,E2 -8714.062} C_VEL
LIN {X 0,Y 446.925,Z 585.114,A -85,B 0,C 180,E1 -8715.895,E2 -8715.895} C_VEL
LIN {X 0,Y 446.353,Z 593.36,A -85,B 0,C 180,E1 -8717.808,E2 -8717.808} C_VEL
LIN {X 0,Y 445.887,Z 599.636,A -85,B 0,C 180,E1 -8719.559,E2 -8719.559} C_VEL
LIN {X 0,Y 445.643,Z 604.959,A -85,B 0,C 180,E1 -8721.386,E2 -8721.386} C_VEL
LIN {X 0,Y 445.567,Z 608.25,A -85,B 0,C 180,E1 -8722.753,E2 -8722.753} C_VEL
LIN {X 0,Y 445.42,Z 611.637,A -85,B 0,C 180,E1 -8724.57,E2 -8724.57} C_VEL
LIN {X 0,Y 445.329,Z 614.093,A -85,B 0,C 180,E1 -8726.383,E2 -8726.383} C_VEL
LIN {X 0,Y 445.346,Z 615.479,A -85,B 0,C 180,E1 -8728.194,E2 -8728.194} C_VEL
LIN {X 0,Y 445.287,Z 616,A -85,B 0,C 180,E1 -8730.002,E2 -8730.002} C_VEL
LIN {X 0,Y 445.346,Z 615.476,A -85,B 0,C 180,E1 -8731.811,E2 -8731.811} C_VEL
LIN {X 0,Y 445.33,Z 614.087,A -85,B 0,C 180,E1 -8733.621,E2 -8733.621} C_VEL
LIN {X 0,Y 445.422,Z 611.629,A -85,B 0,C 180,E1 -8735.434,E2 -8735.434} C_VEL
LIN {X 0,Y 445.571,Z 608.248,A -85,B 0,C 180,E1 -8737.251,E2 -8737.251} C_VEL
LIN {X 0,Y 445.736,Z 602.461,A -85,B 0,C 180,E1 -8739.532,E2 -8739.532} C_VEL
LIN {X 0,Y 446.226,Z 594.847,A -85,B 0,C 180,E1 -8741.817,E2 -8741.817} C_VEL
LIN {X 0,Y 446.768,Z 587.241,A -85,B 0,C 180,E1 -8743.65,E2 -8743.65} C_VEL
LIN {X 0,Y 447.401,Z 579.148,A -85,B 0,C 180,E1 -8745.257,E2 -8745.257} C_VEL
LIN {X 0,Y 448.204,Z 569.594,A -85,B 0,C 180,E1 -8746.857,E2 -8746.857} C_VEL
LIN {X 0,Y 449.221,Z 558.216,A -85,B 0,C 180,E1 -8748.472,E2 -8748.472} C_VEL
LIN {X 0,Y 450.284,Z 545.902,A -85,B 0,C 180,E1 -8749.965,E2 -8749.965} C_VEL
LIN {X 0,Y 451.512,Z 532.612,A -85,B 0,C 180,E1 -8751.338,E2 -8751.338} C_VEL
LIN {X 0,Y 452.754,Z 518.215,A -85,B 0,C 180,E1 -8752.595,E2 -8752.595} C_VEL
LIN {X 0,Y 453.954,Z 504.186,A -85,B 0,C 180,E1 -8753.617,E2 -8753.617} C_VEL
LIN {X 0,Y 454.97,Z 489.733,A -85,B 0,C 180,E1 -8754.493,E2 -8754.493} C_VEL
LIN {X 0,Y 455.986,Z 474.131,A -85,B 0,C 180,E1 -8755.263,E2 -8755.263} C_VEL
LIN {X 0,Y 456.79,Z 458.746,A -85,B 0,C 180,E1 -8755.86,E2 -8755.86} C_VEL
LIN {X 0,Y 457.129,Z 447.444,A -85,B 0,C 180,E1 -8756.195,E2 -8756.195} C_VEL
LIN {X 0,Y 453.316,Z 429.918,A -85,B 0,C 180,E1 -8756.778,E2 -8756.778} C_VEL
LIN {X 0,Y 451.332,Z 418.572,A -85,B 0,C 180,E1 -8757.098,E2 -8757.098} C_VEL
LIN {X 0,Y 452.772,Z 397.545,A -85,B 0,C 180,E1 -8760.556,E2 -8760.556} C_VEL
LIN {X 0,Y 454.476,Z 380.913,A -85,B 0,C 180,E1 -8763.513,E2 -8763.513} C_VEL
LIN {X 0,Y 456.797,Z 365.36,A -85,B 0,C 180,E1 -8766.599,E2 -8766.599} C_VEL
LIN {X 0,Y 457.204,Z 361.977,A -85,B 0,C 180,E1 -8767.387,E2 -8767.387} C_VEL
LIN {X 0,Y 455.766,Z 355.62,A -85,B 0,C 180,E1 -8769.216,E2 -8769.216} C_VEL
LIN {X 0,Y 454.03,Z 349.808,A -85,B 0,C 180,E1 -8771.347,E2 -8771.347} C_VEL
LIN {X 0,Y 452.777,Z 346.053,A -85,B 0,C 180,E1 -8773.153,E2 -8773.153} C_VEL
LIN {X 0,Y 452.104,Z 344.06,A -85,B 0,C 180,E1 -8774.391,E2 -8774.391} C_VEL
LIN {X 0,Y 451.551,Z 342.448,A -85,B 0,C 180,E1 -8775.723,E2 -8775.723} C_VEL
LIN {X 0,Y 450.939,Z 341.009,A -85,B 0,C 180,E1 -8777.921,E2 -8777.921} C_VEL
LIN {X 0,Y 450.676,Z 340.988,A -85,B 0,C 180,E1 -8780.256,E2 -8780.256} C_VEL
LIN {X 0,Y 450.621,Z 342.347,A -85,B 0,C 180,E1 -8782.696,E2 -8782.696} C_VEL
LIN {X 0,Y 450.407,Z 344.415,A -85,B 0,C 180,E1 -8784.737,E2 -8784.737} C_VEL
LIN {X 0,Y 449.616,Z 348.252,A -85,B 0,C 180,E1 -8787.575,E2 -8787.575} C_VEL
LIN {X 0,Y 448.885,Z 353.407,A -85,B 0,C 180,E1 -8790.965,E2 -8790.965} C_VEL
LIN {X 0,Y 448.45,Z 358.257,A -85,B 0,C 180,E1 -8793.972,E2 -8793.972} C_VEL
LIN {X 0,Y 448.086,Z 363.144,A -85,B 0,C 180,E1 -8796.914,E2 -8796.914} C_VEL
LIN {X 0,Y 447.816,Z 368.069,A -85,B 0,C 180,E1 -8799.802,E2 -8799.802} C_VEL
LIN {X 0,Y 447.537,Z 373.096,A -85,B 0,C 180,E1 -8802.696,E2 -8802.696} C_VEL
LIN {X 0,Y 452.415,Z 387.059,A -85,B 0,C 180,E1 -8803.582,E2 -8803.582} C_VEL
LIN {X 0,Y 452.73,Z 389.509,A -85,B 0,C 180,E1 -8803.717,E2 -8803.717} C_VEL
LIN {X 0,Y 452.024,Z 403.043,A -85,B 0,C 180,E1 -8804.443,E2 -8804.443} C_VEL
LIN {X 0,Y 451.281,Z 415.934,A -85,B 0,C 180,E1 -8805.33,E2 -8805.33} C_VEL
LIN {X 0,Y 450.509,Z 427.741,A -85,B 0,C 180,E1 -8806.353,E2 -8806.353} C_VEL
LIN {X 0,Y 449.839,Z 437.396,A -85,B 0,C 180,E1 -8807.366,E2 -8807.366} C_VEL
LIN {X 0,Y 449.289,Z 446.333,A -85,B 0,C 180,E1 -8808.496,E2 -8808.496} C_VEL
LIN {X 0,Y 448.614,Z 455.156,A -85,B 0,C 180,E1 -8809.849,E2 -8809.849} C_VEL
LIN {X 0,Y 448.052,Z 462.77,A -85,B 0,C 180,E1 -8811.314,E2 -8811.314} C_VEL
LIN {X 0,Y 447.49,Z 468.859,A -85,B 0,C 180,E1 -8812.782,E2 -8812.782} C_VEL
LIN {X 0,Y 447.208,Z 473.191,A -85,B 0,C 180,E1 -8814.137,E2 -8814.137} C_VEL
LIN {X 0,Y 447.033,Z 476.441,A -85,B 0,C 180,E1 -8815.492,E2 -8815.492} C_VEL
LIN {X 0,Y 446.89,Z 478.084,A -85,B 0,C 180,E1 -8816.394,E2 -8816.394} C_VEL
LIN {X 0,Y 446.728,Z 479.286,A -85,B 0,C 180,E1 -8817.295,E2 -8817.295} C_VEL
LIN {X 0,Y 446.549,Z 480.075,A -85,B 0,C 180,E1 -8818.197,E2 -8818.197} C_VEL
LIN {X 0,Y 446.497,Z 480.453,A -85,B 0,C 180,E1 -8819.098,E2 -8819.098} C_VEL
LIN {X 0,Y 446.421,Z 480.449,A -85,B 0,C 180,E1 -8820,E2 -8820} C_VEL
LIN {X 0,Y 446.4,Z 480.03,A -85,B 0,C 180,E1 -8820.902,E2 -8820.902} C_VEL
LIN {X 0,Y 446.418,Z 479.177,A -85,B 0,C 180,E1 -8821.805,E2 -8821.805} C_VEL
LIN {X 0,Y 446.512,Z 477.921,A -85,B 0,C 180,E1 -8822.707,E2 -8822.707} C_VEL
LIN {X 0,Y 446.514,Z 475.284,A -85,B 0,C 180,E1 -8824.062,E2 -8824.062} C_VEL
LIN {X 0,Y 446.513,Z 471.659,A -85,B 0,C 180,E1 -8825.419,E2 -8825.419} C_VEL
LIN {X 0,Y 446.857,Z 466.916,A -85,B 0,C 180,E1 -8826.775,E2 -8826.775} C_VEL
LIN {X 0,Y 447.102,Z 459.889,A -85,B 0,C 180,E1 -8828.361,E2 -8828.361} C_VEL
LIN {X 0,Y 447.519,Z 452.314,A -85,B 0,C 180,E1 -8829.72,E2 -8829.72} C_VEL
LIN {X 0,Y 447.911,Z 442.988,A -85,B 0,C 180,E1 -8831.082,E2 -8831.082} C_VEL
LIN {X 0,Y 448.527,Z 432.485,A -85,B 0,C 180,E1 -8832.327,E2 -8832.327} C_VEL
LIN {X 0,Y 449.032,Z 420.644,A -85,B 0,C 180,E1 -8833.463,E2 -8833.463} C_VEL
LIN {X 0,Y 449.557,Z 408.397,A -85,B 0,C 180,E1 -8834.407,E2 -8834.407} C_VEL
LIN {X 0,Y 450.13,Z 395.916,A -85,B 0,C 180,E1 -8835.161,E2 -8835.161} C_VEL
LIN {X 0,Y 450.39,Z 383.696,A -85,B 0,C 180,E1 -8835.737,E2 -8835.737} C_VEL
LIN {X 0,Y 446.979,Z 369.464,A -85,B 0,C 180,E1 -8836.371,E2 -8836.371} C_VEL
LIN {X 0,Y 446.113,Z 365.883,A -85,B 0,C 180,E1 -8836.503,E2 -8836.503} C_VEL
LIN {X 0,Y 446.192,Z 360.338,A -85,B 0,C 180,E1 -8839.316,E2 -8839.316} C_VEL
LIN {X 0,Y 446.318,Z 354.696,A -85,B 0,C 180,E1 -8842.205,E2 -8842.205} C_VEL
